   - Come identifico l'assenza del nodo?? (Rele non funzionante/non alimentato)
   - Acquisizione carico dopo accensione?? Dati carico in NVM!
   
   v1.0[07/05/15] - Create
*)
VAR CONSTANT
	MANUAL			: BYTE := 0;
	AUTOMATIC		: BYTE := 1;
	SCHEDULED		: BYTE := 2;
END_VAR
VAR_INPUT
	(* Settings *)
	ID				: BYTE;
	(* Controls *)
	CTRL_MODE		: BYTE;  (* 0 : MANUAL, (human) user manage the lux						->	HIGHEST PRIORITY
							    1 : AUTO, external device/sensor manage the lux				->	MID PRIORITY
							    2 : SCHEDULED, scheduled profile with crono manage the lux	->	LOWEST PRIORITY
							  *)

	(* Forced inputs *)
	LUX_ON_REQ		: BOOL; (* On request (Only "LUX_OFF_REQ" has highest priority) *)
	LUX_OFF_REQ		: BOOL; (* Off request (Highest priority over all other inputs/commands) *)

	(* External physical/software inputs *)
	CTRL_KEY		: BOOL := FALSE; (* External KEY control input *)
	KEY_PUSH		: BOOL := FALSE; (* 0: key as latch switch, 1: key as push-button, changes output state every time  *)
	CTRL_EXT_DS		: BOOL := FALSE; (* External DEVICE/SENSOR input *)
	CTRL_CRON		: BOOL := FALSE; (* External forced activation *)

	(* Conditional event *)
	CTRL_COND		: typ_Condition;
	CTRL_AUTO		: BOOL := TRUE;		(* 1: Lux managed by plc, 0: plc by-passed, managed by user	*)
	SINGLE_FEEDBACK	: BOOL;			 	(* Lux has its own feedback to control output status (state of art) or a general
										   feedback shared with other lux (loss of precision) *)

	(* Physical inputs (feedback) *)
	OUT_ST			: BOOL; (* Status feedback *)

END_VAR
VAR_IN_OUT
	WORKINGTIME		: DWORD; (* [sec] Internal working time counter *)
	POWERONCYCLES	: DWORD; (* Internal counter of power-on cycles *)
END_VAR
VAR_OUTPUT
	(* Physical outputs *)
	OUT_EN			: BOOL;	(* Control output *)
	(* Status *)
	Status_Log		: BYTE;
	Status_Vis 		: DWORD;
END_VAR
VAR
	InitOK			: BOOL;
	CTRL_MODE_Default: BYTE;
	Force			: BOOL := FALSE;		(* Force output to a value without considering its normal operation	*)

	KeyPress		: FLT_TIME 	:= (INITEV:=FALSE, TTAP:=T#5ms);
	AutoEn			: FLT_TAP := (INITEV:=FALSE);
	sOUT_EN			: FLT_EVENT;

	TickTimer		: TON := ( PT:=T#1s );
	chkOUT_ST		: FLT_TIME := ( TTAP:=T#5s);

	actualTime		: STRING;


END_VAR
Init();

(* Check if one or more conditional events are setted for this LUX *)
Condition();

IF LUX_OFF_REQ THEN OUT_EN := FALSE;
ELSIF LUX_ON_REQ OR NOT CTRL_AUTO THEN OUT_EN := TRUE;
ELSE
	(* Do actions according to acutal working mode *)
	CASE CTRL_MODE OF

		MANUAL:	(* Lux switching is managed by user	*)
	
			KeyPress(IN:=CTRL_KEY);
	
			IF KEY_PUSH THEN
				IF KeyPress.EVH THEN OUT_EN := NOT OUT_EN; END_IF	(* Key as push-button  ->  Toggle output *)
			ELSE
				IF KeyPress.EVH OR KeyPress.EVL THEN OUT_EN := CTRL_KEY; END_IF	(* Key as switch  ->  Open-Switch off
																									  Close-Switch on	*)
			END_IF

	
		AUTOMATIC:	(* Lux managed by an external device/sensor	*)

			KeyPress(IN:=CTRL_KEY);



			(* If a change in the key state has occured, switch to manual mode	*)
			IF KEY_PUSH THEN
				IF KeyPress.EVH THEN
					OUT_EN := NOT OUT_EN; 	(* Toggle output *)
					CTRL_MODE := MANUAL;
				END_IF
			ELSE
				IF KeyPress.EVH OR KeyPress.EVL THEN
					OUT_EN := CTRL_KEY;
					CTRL_MODE := MANUAL;
				END_IF
			END_IF

			(* These instructions are used to manage conditional event *)
			IF CTRL_MODE<>MANUAL THEN
				(* If not Forced keep automatic control *)
				IF NOT Force THEN
					(* Automatic mode *)
					AutoEn(IN:=CTRL_EXT_DS);
	
					(* IF AutoEn.EVH OR AutoEn.EVL THEN OUT_EN := NOT OUT_EN; END_IF *)
					IF AutoEn.EVH THEN OUT_EN := TRUE; END_IF
					IF AutoEn.EVL THEN OUT_EN := FALSE; END_IF
				END_IF
			END_IF

		SCHEDULED:
			(* Check if key has changed its state	*)
			KeyPress(IN:=CTRL_KEY);
	
			IF KEY_PUSH THEN
				IF KeyPress.EVH THEN
					OUT_EN := NOT OUT_EN; 	(* Toggle output *)
					CTRL_MODE := MANUAL;
				END_IF
			ELSE
				IF KeyPress.EVH OR KeyPress.EVL THEN
					OUT_EN := CTRL_KEY;
					CTRL_MODE := MANUAL;
				END_IF
			END_IF
	
			IF CTRL_MODE<>MANUAL THEN
				(* If not forced keep normal control *)
				IF NOT Force THEN
					(* Check if external control device has changed its state	*)
					AutoEn(IN:=CTRL_EXT_DS);
	
					IF AutoEn.EVH OR AutoEn.EVL THEN
						CTRL_MODE := AUTOMATIC;
						OUT_EN := NOT OUT_EN;
					END_IF
	
					IF CTRL_MODE<>AUTOMATIC THEN OUT_EN := CTRL_CRON;	END_IF	(* Scheduled mode	*)
				END_IF
			END_IF

	END_CASE
END_IF

(* Power on cycles and working time counters *)
Counters();

(* Check status feedback *)
IF SINGLE_FEEDBACK THEN chkOUT_ST(IN:=(OUT_ST<>OUT_EN));	(* External status feedback input available *)
ELSE chkOUT_ST(IN:=OUT_ST);						(* No external status feedback *)
END_IF
IF chkOUT_ST.EVH THEN LogEv(EL_Alarm,EO_LUX,ID,9,''); END_IF
IF chkOUT_ST.EVL THEN LogEv(EL_Log,EO_LUX,ID,1,''); END_IF

(* Status color *)
IF chkOUT_ST.OUT	THEN Status_Log:=2; (*Status_Vis:=COLOR_RED;*)
ELSE Status_Log:=0; Status_Vis:=SEL(OUT_EN,COLOR_GREEN_OFF,COLOR_GREEN);
END_IF
END_FUNCTION_BLOCK
ACTION AddLogData:
Logger.s1:=INSERT('&LUX=',BYTE_TO_STRING(ID),4);
IF ID<10 THEN Logger.s1:=INSERT(Logger.s1,'0',4); END_IF

Logger.s1:=CONCAT(Logger.s1,BOOL_TO_STRING(OUT_EN));			Logger.s1:=CONCAT(Logger.s1,';');
Logger.s1:=CONCAT(Logger.s1,DWORD_TO_STRING(WORKINGTIME));		Logger.s1:=CONCAT(Logger.s1,';');
Logger.s1:=CONCAT(Logger.s1,DWORD_TO_STRING(POWERONCYCLES));	Logger.s1:=CONCAT(Logger.s1,';');
Logger.s1:=CONCAT(Logger.s1,BYTE_TO_STRING(CTRL_MODE));			Logger.s1:=CONCAT(Logger.s1,';');
Logger.s1:=CONCAT(Logger.s1,BYTE_TO_STRING(Status_Log));
Logger.s1:=CONCAT(Logger.s1,';');
Logger.s1:=CONCAT(Logger.s1,SEL(LUX_ON_REQ,'0','100'));
Logger.s1:=CONCAT(Logger.s1,';');
Logger.s1:=CONCAT(Logger.s1,SEL(LUX_OFF_REQ,'0','100'));




ADDSTRING(ADR(Logger.TData), ADR(Logger.s1), Logger.TLen);
END_ACTION
ACTION Condition:
CASE CTRL_COND.Enable OF

	0:	(* NO CONDITION	*)
		;

	1:	(* BOOLEAN CONDITION - Trig On *)
		IF CTRL_COND.OnIN=CTRL_COND.OnValue THEN OUT_EN:=TRUE; END_IF

	2:	(* BOOLEAN CONDITION - Trig Off *)
		IF CTRL_COND.OffIN=CTRL_COND.OffValue THEN OUT_EN:=FALSE; END_IF

	3:	(* BOOLEAN CONDITION - Trig On and Off *)
		IF (OUT_EN=FALSE AND CTRL_COND.OnIN=CTRL_COND.OnValue) THEN OUT_EN:=TRUE; END_IF
		IF (OUT_EN=TRUE AND CTRL_COND.OffIN=CTRL_COND.OffValue) THEN OUT_EN:=FALSE; END_IF

	4: 	(* TIME of DAY - Trig On *)
		actualTime := MID(STR:=Sys.Time_LogString, LEN:=5, POS:=12);		(* Check if time of the day reached *)

		IF (OUT_EN=FALSE AND actualTime>=TOD_TO_STRING(CTRL_COND.OnTime)) THEN OUT_EN:=TRUE; END_IF

	5: 	(* TIME of DAY - Trig Off *)
		actualTime := MID(STR:=Sys.Time_LogString, LEN:=5, POS:=12);

		IF (OUT_EN=TRUE AND actualTime>=TOD_TO_STRING(CTRL_COND.OffTime)) THEN
			OUT_EN:= FALSE;
			Force := TRUE;
		END_IF

		IF actualTime>='08:00' THEN Force := FALSE; END_IF	(* Release force and restore normal working *)

END_CASE
END_ACTION
ACTION Counters:
(* Temporary energy counter *)
TickTimer(IN:=NOT TickTimer.Q);
IF (TickTimer.Q AND OUT_EN) THEN WORKINGTIME:=WORKINGTIME+1; END_IF

(* Generate status events *)
sOUT_EN(IN:=OUT_EN);
IF sOUT_EN.EVL THEN LogEv(EL_Log,EO_LUX,ID,2,''); END_IF
IF sOUT_EN.EVH THEN LogEv(EL_Log,EO_LUX,ID,3,''); POWERONCYCLES:=POWERONCYCLES+1; END_IF
END_ACTION
ACTION Init:
IF NOT InitOK THEN
	(* First time read the CTRL_MODE setted by the programmer in the global variables definition *)
	CTRL_MODE_Default := CTRL_MODE;
	InitOK := TRUE;
END_IF
END_ACTION
ACTION RestoreMode:
CTRL_MODE := CTRL_MODE_Default;

LUX_ON_REQ := FALSE;
LUX_OFF_REQ:= FALSE;
END_ACTION
ACTION StatReset:
(* Reset statistic counters *)
WORKINGTIME:=0;
POWERONCYCLES:=0;
END_ACTION

(* POU Plant_Objects/obj_MODBUS_FRER_QUBOH, ST *)
FUNCTION_BLOCK obj_MODBUS_FRER_QUBOH
(* === MODBUS ELECTRICITY CONTABILIZER ABB ===
   v1.0[20/08/15] - Versioning
*)
VAR CONSTANT
	WAIT_STATE		:	BYTE := 0;
	START_READ		:	BYTE := 1;
	READ_1			:	BYTE := 2;
	READ_2			:	BYTE := 3;
	READ_3			:	BYTE := 4;
	READ_4			:	BYTE := 5;
	READ_5			:	BYTE := 6;
	END_READ		:	BYTE := 7;
	WRITE_Q			:	BYTE := 8;
	READ_6			:	BYTE := 9;
	WRITE_ENABLE	:	BYTE := 10;

	ERROR_STATE		:	BYTE := 100;
END_VAR
VAR_INPUT
	ID				:	BYTE;
	Address			:	BYTE;

	Refresh_Period	: 	TIME:=t#1m;
	(* Controls *)
	Refresh_Auto	: 	BOOL:=TRUE; (* Enable automatic refresh *)
	Refresh_Now		:	BOOL; 	  (* Force an immediate refresh *)
END_VAR
VAR_IN_OUT
	ModBus		:	obj_MODBUS;
END_VAR
VAR_OUTPUT
	Status_Log	:	WORD;
	Status_Vis	:	DWORD;
END_VAR
VAR
	Data		:	typ_MODBUS_FRER_QUBOH;

	WH_3P		:	DWORD;		(* E-1 kWh *)
	VARH_3P		:	DWORD;		(* E-1 kVArh *)

	Q_Max		:	DWORD;

	dly 		: 	TON := (PT:=t#5s);
	state		: 	BYTE; 	(* Status *)
	retry		: 	BYTE;
END_VAR
CASE state OF

	WAIT_STATE: (* === Wait update signals *)
		dly(IN:=NOT (dly.Q OR Refresh_Now OR (NOT Refresh_Auto)));
		IF dly.Q OR Refresh_Now THEN
			dly.PT := Refresh_Period;
			Refresh_Now := FALSE;
			state := START_READ;
		END_IF

	START_READ:(* === Start update when MB is free *)
		IF NOT (ModBus.MB_Lock OR ModBus.MB_Start) THEN

			ModBus.MB_Lock := TRUE;
			ModBus.MB_Query.SlaveAddress := Address;
			ModBus.MB_Query.FunctionCode := 16#03;
			(* Start query *)
			ModBus.MB_Query.Read_StartAddress := 16#0100;
			ModBus.MB_Query.Read_Quantity := 32;
			ModBus.MB_Start := TRUE;

			state := READ_1;
		END_IF

	READ_1:
		IF NOT ModBus.MB_Start THEN
			IF ModBus.MB_MASTER.MB_Error<>MB_NO_ERROR OR ModBus.MB_Resp.Error<>0 THEN
				state := ERROR_STATE;
			ELSE
				(* Read response data *)
				COPY_32SWAP16(ADR(ModBus.MB_Resp.Data[0]), ADR(Data.V_L1N));
				COPY_32SWAP16(ADR(ModBus.MB_Resp.Data[2]), ADR(Data.V_L2N));
				COPY_32SWAP16(ADR(ModBus.MB_Resp.Data[4]), ADR(Data.V_L3N));
				COPY_32SWAP16(ADR(ModBus.MB_Resp.Data[6]), ADR(Data.V_L1L2));
				COPY_32SWAP16(ADR(ModBus.MB_Resp.Data[8]), ADR(Data.V_L2L3));
				COPY_32SWAP16(ADR(ModBus.MB_Resp.Data[10]), ADR(Data.V_L3L1));
				COPY_32SWAP16(ADR(ModBus.MB_Resp.Data[12]), ADR(Data.I_L1));
				COPY_32SWAP16(ADR(ModBus.MB_Resp.Data[14]), ADR(Data.I_L2));
				COPY_32SWAP16(ADR(ModBus.MB_Resp.Data[16]), ADR(Data.I_L3));
				COPY_32SWAP16(ADR(ModBus.MB_Resp.Data[18]), ADR(Data.FREQ));
				COPY_32SWAP16(ADR(ModBus.MB_Resp.Data[20]), ADR(Data.P_3P));
				COPY_32SWAP16(ADR(ModBus.MB_Resp.Data[22]), ADR(Data.Q_3P));
				COPY_32SWAP16(ADR(ModBus.MB_Resp.Data[24]), ADR(Data.PF_3P));
				COPY_32SWAP16(ADR(ModBus.MB_Resp.Data[26]), ADR(Data.WH_3P));
				COPY_32SWAP16(ADR(ModBus.MB_Resp.Data[28]), ADR(Data.VARH_3P));
				COPY_32SWAP16(ADR(ModBus.MB_Resp.Data[30]), ADR(Data.Multiplier));

				(* Evaluate energy according to read multiplier factor *)
				WH_3P := (Data.WH_3P * Data.Multiplier)/100;		(* Divided by 100 because read value is in Wh, we need E-1 kWh *)
				VARH_3P := (Data.VARH_3P * Data.Multiplier)/100;

				ModBus.MB_Query.Read_StartAddress := 16#0122;
				ModBus.MB_Query.Read_Quantity := 4;
				ModBus.MB_Start := TRUE;

				state := READ_2;
			END_IF
		END_IF

	READ_2:
		IF NOT ModBus.MB_Start THEN
			IF ModBus.MB_MASTER.MB_Error<>MB_NO_ERROR OR ModBus.MB_Resp.Error<>0 THEN
				state := ERROR_STATE;
			ELSE
				(* Read response data *)
				COPY_32SWAP16(ADR(ModBus.MB_Resp.Data[0]), ADR(Data.V_3P));
				COPY_32SWAP16(ADR(ModBus.MB_Resp.Data[2]), ADR(Data.I_3P));

				ModBus.MB_Query.Read_StartAddress := 16#012E;
				ModBus.MB_Query.Read_Quantity := 2;
				ModBus.MB_Start := TRUE;

				state := READ_3;
			END_IF
		END_IF

	READ_3:
		IF NOT ModBus.MB_Start THEN
			IF ModBus.MB_MASTER.MB_Error<>MB_NO_ERROR OR ModBus.MB_Resp.Error<>0 THEN
				state := ERROR_STATE;
			ELSE
				(* Read response data *)
				COPY_32SWAP16(ADR(ModBus.MB_Resp.Data[0]), ADR(Data.COS_3P));

				ModBus.MB_Query.Read_StartAddress := 16#0142;
				ModBus.MB_Query.Read_Quantity := 20;
				ModBus.MB_Start := TRUE;

				state := READ_4;
			END_IF
		END_IF

	READ_4:
		IF NOT ModBus.MB_Start THEN
			IF ModBus.MB_MASTER.MB_Error<>MB_NO_ERROR OR ModBus.MB_Resp.Error<>0 THEN
				state := ERROR_STATE;
			ELSE
				COPY_32SWAP16(ADR(ModBus.MB_Resp.Data[0]), ADR(Data.VA_3P));
				COPY_32SWAP16(ADR(ModBus.MB_Resp.Data[2]), ADR(Data.P_L1));
				COPY_32SWAP16(ADR(ModBus.MB_Resp.Data[4]), ADR(Data.P_L2));
				COPY_32SWAP16(ADR(ModBus.MB_Resp.Data[6]), ADR(Data.P_L3));
				COPY_32SWAP16(ADR(ModBus.MB_Resp.Data[8]), ADR(Data.Q_L1));
				COPY_32SWAP16(ADR(ModBus.MB_Resp.Data[10]), ADR(Data.Q_L2));
				COPY_32SWAP16(ADR(ModBus.MB_Resp.Data[12]), ADR(Data.Q_L3));
				COPY_32SWAP16(ADR(ModBus.MB_Resp.Data[14]), ADR(Data.VA_L1));
				COPY_32SWAP16(ADR(ModBus.MB_Resp.Data[16]), ADR(Data.VA_L2));
				COPY_32SWAP16(ADR(ModBus.MB_Resp.Data[18]), ADR(Data.VA_L3));

				ModBus.MB_Query.Read_StartAddress := 16#0156;
				ModBus.MB_Query.Read_Quantity := 22;
				ModBus.MB_Start := TRUE;

				state := READ_5;
			END_IF
		END_IF

	READ_5:
		IF NOT ModBus.MB_Start THEN
			IF ModBus.MB_MASTER.MB_Error<>MB_NO_ERROR OR ModBus.MB_Resp.Error<>0 THEN
				state := ERROR_STATE;
			ELSE
				COPY_32SWAP16(ADR(ModBus.MB_Resp.Data[0]), ADR(Data.PF_L1));
				COPY_32SWAP16(ADR(ModBus.MB_Resp.Data[2]), ADR(Data.PF_L2));
				COPY_32SWAP16(ADR(ModBus.MB_Resp.Data[4]), ADR(Data.PF_L3));
				COPY_32SWAP16(ADR(ModBus.MB_Resp.Data[6]), ADR(Data.COS_L1));
				COPY_32SWAP16(ADR(ModBus.MB_Resp.Data[8]), ADR(Data.COS_L2));
				COPY_32SWAP16(ADR(ModBus.MB_Resp.Data[10]), ADR(Data.COS_L3));
				COPY_32SWAP16(ADR(ModBus.MB_Resp.Data[12]), ADR(Data.P_3P_Max));
				COPY_32SWAP16(ADR(ModBus.MB_Resp.Data[14]), ADR(Data.P_3P_Avg));
				COPY_32SWAP16(ADR(ModBus.MB_Resp.Data[16]), ADR(Data.I_L1_Max));
				COPY_32SWAP16(ADR(ModBus.MB_Resp.Data[18]), ADR(Data.I_L2_Max));
				COPY_32SWAP16(ADR(ModBus.MB_Resp.Data[20]), ADR(Data.I_L3_Max));

				ModBus.MB_Query.Read_StartAddress := 16#01A6;
				ModBus.MB_Query.Read_Quantity := 2;
				ModBus.MB_Start := TRUE;

				state := END_READ;
			END_IF
		END_IF

	END_READ:
		IF NOT ModBus.MB_Start THEN
			IF ModBus.MB_MASTER.MB_Error<>MB_NO_ERROR OR ModBus.MB_Resp.Error<>0 THEN
				state := ERROR_STATE;
			ELSE
				COPY_32SWAP16(ADR(ModBus.MB_Resp.Data[0]), ADR(Data.Q_3P_Max));

				ModBus.MB_Query.Write_StartAddress := 16#200;
				ModBus.MB_Query.FunctionCode := 16#10;
				ModBus.MB_Query.Write_Quantity := 2;
				ModBus.MB_Query.Write_Data[0] := 16#0000;
				ModBus.MB_Query.Write_Data[1] := 16#00A5;
				ModBus.MB_Start := TRUE;

				state := WRITE_ENABLE;
			END_IF
		END_IF

	WRITE_ENABLE:
		IF NOT ModBus.MB_Start THEN
			IF ModBus.MB_MASTER.MB_Error<>MB_NO_ERROR OR ModBus.MB_Resp.Error<>0 THEN
				state := ERROR_STATE;
			ELSE
				COPY_32SWAP16(ADR(ModBus.MB_Resp.Data[0]), ADR(Data.Q_3P_Max));

				ModBus.MB_Query.Write_StartAddress := 16#01A6;
				ModBus.MB_Query.FunctionCode := 16#10;
				ModBus.MB_Query.Write_Quantity := 2;
				ModBus.MB_Query.Write_Data[0] := 16#0000;
				ModBus.MB_Query.Write_Data[1] := 16#0000;
				ModBus.MB_Start := TRUE;

				state := WRITE_Q;
			END_IF
		END_IF

	WRITE_Q:
		IF NOT ModBus.MB_Start THEN
			IF ModBus.MB_MASTER.MB_Error<>MB_NO_ERROR OR ModBus.MB_Resp.Error<>0 THEN
				state := ERROR_STATE;
			ELSE
				ModBus.MB_Query.Read_StartAddress := 16#01A6;
				ModBus.MB_Query.FunctionCode := 16#03;
				ModBus.MB_Query.Read_Quantity := 2;

				ModBus.MB_Start := TRUE;
				state := READ_6;
			END_IF
		END_IF

	READ_6:
		IF NOT ModBus.MB_Start THEN
			IF ModBus.MB_MASTER.MB_Error<>MB_NO_ERROR OR ModBus.MB_Resp.Error<>0 THEN
				state := ERROR_STATE;
			ELSE
				COPY_32SWAP16(ADR(ModBus.MB_Resp.Data[0]), ADR(Q_Max));
				(* Signal event *)
				(*IF Status_Log<>0 THEN
					LogEv(EL_Log,EO_ANZ,ID,1,'');
				END_IF*)

				(* Update status *)
				Status_Log:=0;

				ModBus.MB_Lock := FALSE;
				retry := 0;
				state := WAIT_STATE;
			END_IF
		END_IF

	ERROR_STATE: (* === Check MODBUS error *)
			(* Release MODBUS *)
			MODBUS.MB_Lock:=FALSE;

			(* Retries *)
			retry:=retry+1;

			IF retry>3 THEN
				retry:=0;
				(* Signal event *)
				IF Status_Log<>2 THEN
					LogEv(EL_Alarm,EO_ANZ,ID,2,SEL(ModBus.MB_MASTER.MB_Error<>0,'0','1'));
				END_IF
				(* Update status *)
				Status_Log:=2;
			END_IF

			state := WAIT_STATE;

END_CASE

IF Status_Log=2 THEN Status_Vis := COLOR_RED;
ELSE Status_Vis := COLOR_GREEN;
END_IF
END_FUNCTION_BLOCK
ACTION AddLogData:
Logger.s1:=INSERT('&ANZ=',BYTE_TO_STRING(ID),4);
IF ID<10 THEN Logger.s1:=INSERT(Logger.s1,'0',4); END_IF

Logger.s1:=CONCAT(Logger.s1,DWORD_TO_STRING(Data.V_L1N/1000));		Logger.s1:=CONCAT(Logger.s1,';');
Logger.s1:=CONCAT(Logger.s1,DWORD_TO_STRING(Data.V_L2N/1000));		Logger.s1:=CONCAT(Logger.s1,';');
Logger.s1:=CONCAT(Logger.s1,DWORD_TO_STRING(Data.V_L3N/1000));		Logger.s1:=CONCAT(Logger.s1,';');
Logger.s1:=CONCAT(Logger.s1,DWORD_TO_STRING(Data.V_L1L2/1000));		Logger.s1:=CONCAT(Logger.s1,';');
Logger.s1:=CONCAT(Logger.s1,DWORD_TO_STRING(Data.V_L2L3/1000));		Logger.s1:=CONCAT(Logger.s1,';');
Logger.s1:=CONCAT(Logger.s1,DWORD_TO_STRING(Data.V_L3L1/1000));		Logger.s1:=CONCAT(Logger.s1,';');

Logger.s1:=CONCAT(Logger.s1,DWORD_TO_STRING(Data.FREQ));		Logger.s1:=CONCAT(Logger.s1,';');

Logger.s1:=CONCAT(Logger.s1,DWORD_TO_STRING(Data.I_L1));		Logger.s1:=CONCAT(Logger.s1,';');
Logger.s1:=CONCAT(Logger.s1,DWORD_TO_STRING(Data.I_L2));		Logger.s1:=CONCAT(Logger.s1,';');
Logger.s1:=CONCAT(Logger.s1,DWORD_TO_STRING(Data.I_L3));		Logger.s1:=CONCAT(Logger.s1,';');
Logger.s1:=CONCAT(Logger.s1,DWORD_TO_STRING(Data.I_L1_Max)); 	Logger.s1:=CONCAT(Logger.s1,';');
Logger.s1:=CONCAT(Logger.s1,DWORD_TO_STRING(Data.I_L2_Max)); 	Logger.s1:=CONCAT(Logger.s1,';');
Logger.s1:=CONCAT(Logger.s1,DWORD_TO_STRING(Data.I_L3_Max)); 	Logger.s1:=CONCAT(Logger.s1,';');

Logger.s1:=CONCAT(Logger.s1,DINT_TO_STRING(Data.PF_L1));		Logger.s1:=CONCAT(Logger.s1,';');
Logger.s1:=CONCAT(Logger.s1,DINT_TO_STRING(Data.PF_L2));		Logger.s1:=CONCAT(Logger.s1,';');
Logger.s1:=CONCAT(Logger.s1,DINT_TO_STRING(Data.PF_L3));		Logger.s1:=CONCAT(Logger.s1,';');

Logger.s1:=CONCAT(Logger.s1,DWORD_TO_STRING(Data.P_3P));		Logger.s1:=CONCAT(Logger.s1,';');
Logger.s1:=CONCAT(Logger.s1,DWORD_TO_STRING(Data.P_3P_Avg)); 	Logger.s1:=CONCAT(Logger.s1,';');
Logger.s1:=CONCAT(Logger.s1,DWORD_TO_STRING(Data.P_3P_Max)); 	Logger.s1:=CONCAT(Logger.s1,';');

Logger.s1:=CONCAT(Logger.s1,DINT_TO_STRING(Data.Q_3P));			Logger.s1:=CONCAT(Logger.s1,';');
Logger.s1:=CONCAT(Logger.s1,DINT_TO_STRING(Data.Q_3P_Max));		Logger.s1:=CONCAT(Logger.s1,';');

Logger.s1:=CONCAT(Logger.s1,DWORD_TO_STRING(WH_3P));			Logger.s1:=CONCAT(Logger.s1,';');
Logger.s1:=CONCAT(Logger.s1,DWORD_TO_STRING(VARH_3P));			Logger.s1:=CONCAT(Logger.s1,';');

Logger.s1:=CONCAT(Logger.s1,WORD_TO_STRING(Status_Log));
ADDSTRING(ADR(Logger.TData), ADR(Logger.s1), Logger.TLen);
END_ACTION

(* POU Plant_Objects/obj_MODBUS_TCP, ST *)
FUNCTION_BLOCK obj_MODBUS_TCP
(* === MODBUS-TCP PROTOCOL INTERFACE ===
   v1.0[10/06/15] - Create
*)
VAR CONSTANT
	VARS_Max	: BYTE := 32;
END_VAR
VAR_INPUT
	(* Settings *)
	ID			: BYTE;
	IP			: STRING;
	PORT		: WORD:=502;
	(* Interface *)
	MB_MASTER	: ETHERNET_MODBUSMASTER_TCP;
	MB_READBUF	: ARRAY [0..128] OF WORD;
	MB_WRITEBUF : ARRAY [0..128] OF WORD;
	MB_Start	: BOOL;
	MB_Lock		: BOOL;
	(* Variables management *)
	VARS_En		: BOOL;
	VARS		: ARRAY [0..VARS_Max] OF typ_MODBUS_VAR;
	VARS_Check	: BOOL;
	VARS_Alarm	: BOOL;
	(* Variables allocation *)
	VAR_Pointer : POINTER TO ARRAY[0..99] OF WORD;
	VAR_Cfg		: POINTER TO typ_MODBUS_VAR;
END_VAR
VAR_OUTPUT
	(* Status *)
	Status_Log	: BYTE;
	Status_Vis	: DWORD;
END_VAR
VAR
	sta         : BYTE :=0;
	i			: BYTE;
	j			: BYTE;
	Alarm		: FLT_EVENT := (INITEV:=FALSE);

	VarTmr		: TON := (PT:=T#1s);
	VarSta		: BYTE; (* Status *)
	VarCnt		: BYTE; (* Scan counter *)
	VarRetry	: BYTE;
	VarAlarm	: BYTE; (* Last variable with errors *)
END_VAR
MB_MASTER( strIP_ADDRESS:=IP, wPORT:=PORT, tTIME_OUT:=T#750MS, (*xCONNECT:=TRUE,*)
		   ptREAD_DATA:=ADR(MB_READBUF), ptSEND_DATA:=ADR(MB_WRITEBUF), xSEND:=MB_Start );

IF sta=0 THEN
	MB_MASTER.xCONNECT:=TRUE;
	sta:=1;
END_IF

(* Process variable management *)
IF VARS_En THEN VARS_Process(); END_IF

(* Check status *)
Alarm(IN:=(MB_MASTER.wERROR<>0));
IF Alarm.EVH THEN
	LogEv(SEL(MB_MASTER.wERROR>0,EL_Wrn,EL_Alarm),EO_MODBUS_TCP,ID,1,WORD_TO_STRING(MB_MASTER.wERROR));
END_IF
IF Alarm.EVL THEN
	LogEv(EL_Log,EO_MODBUS_TCP,ID,2,'');
END_IF

(* Log/visu status *)
   IF Alarm.IN   THEN Status_Log:=2; Status_Vis:=COLOR_RED;
ELSIF Vars_Alarm THEN Status_Log:=1; Status_Vis:=COLOR_YELLOW;
  				 ELSE Status_Log:=0; Status_Vis:=COLOR_GREEN;
END_IF
END_FUNCTION_BLOCK
ACTION VAR_Search:
(* Search VAR with specific pointer if not found return first free VAR
	[Last VAR is not active... used as safe area...] 
*)
j:=VARS_Max;
FOR i := 0 TO VARS_Max-1 DO
	IF VARS[i].Variable=0 AND j>i THEN j:=i; END_IF
	IF VARS[i].Variable=VAR_Pointer THEN
		VAR_Cfg:=ADR(VARS[i]);
		RETURN;
	END_IF
END_FOR
VAR_Cfg:=ADR(VARS[j]);
END_ACTION
ACTION VARS_Process:
(* Update var timers *)
VarTmr(IN:=(NOT VarTmr.Q));
IF VarTmr.Q THEN
	FOR i := 0 TO VARS_Max DO
		IF VARS[i].Refresh_Cnt>0 THEN VARS[i].Refresh_Cnt:=VARS[i].Refresh_Cnt-1; END_IF
	END_FOR
	VARS_Check:=TRUE;
END_IF


(* Process status *)
CASE VarSta OF
	0: (* === Init *)
		VarCnt:=0;
		VarSta:=1;

	1: (* === Wait check signal *)
		IF VARS_Check THEN
			VARS_Check:=FALSE;
			VarCnt:=0;
			VarSta:=2;
		END_IF

	2: (* === Check loop *)
		IF NOT (MB_Lock OR MB_Start) THEN
			WHILE VarCnt<=(VARS_Max-1) AND VarSta=2 DO
				(* Check only active vars *)
				IF VARS[VarCnt].Variable<>0 THEN
					(* Check var auto-refresh on timer checks *)
					IF VARS[VarCnt].Refresh_Time>0 AND VARS[VarCnt].Refresh_Cnt=0 THEN
						VARS[VarCnt].Refresh_Cnt:=VARS[VarCnt].Refresh_Time;
						VarSta:=3;
					END_IF
					(* Check refresh for change or request *)
					CASE VARS[VarCnt].FunCode OF
						5,6,15,16: (* Write functions *)
							IF VARS[VarCnt].Variable_Size=1 THEN
								IF VARS[VarCnt].Variable^<>VARS[VarCnt].Variable_Mirror THEN
									VARS[VarCnt].Variable_Mirror:=VARS[VarCnt].Variable^;
									VarSta:=3;
								END_IF
							ELSE
								IF VARS[VarCnt].Variable_Mirror<>0 THEN
									VARS[VarCnt].Variable_Mirror:=0;
									VarSta:=3;
								END_IF
							END_IF
						1,2,3,4: (* Write functions *)
							IF VARS[VarCnt].Variable_Mirror<>0 THEN
								VARS[VarCnt].Variable_Mirror:=0;
								VarSta:=3;
							END_IF
					END_CASE
				END_IF
				(* Process query *)
				IF VarSta=3 THEN
					MB_Lock:=TRUE;
					MB_MASTER.bUNIT_ID:=VARS[VarCnt].SlaveAddress;
					MB_MASTER.bFUNCTION_CODE:=VARS[VarCnt].FunCode;
					CASE VARS[VarCnt].FunCode OF
						16#5,16#6,16#F,16#10:
							MB_MASTER.wREAD_ADDRESS:=0;
							MB_MASTER.wREAD_QUANTITY:=0;
							MB_MASTER.wWRITE_ADDRESS:=VARS[VarCnt].FunAddress;
							MB_MASTER.wWRITE_QUANTITY:=VARS[VarCnt].Variable_Size;
							IF VARS[VarCnt].Variable_Size=200 THEN
								COPY_32SWAP16(VARS[VarCnt].Variable, ADR(MB_WRITEBUF));
							ELSIF VARS[VarCnt].Variable_Size>1 THEN
								MEMCPY(VARS[VarCnt].Variable, ADR(MB_WRITEBUF), 2*VARS[VarCnt].Variable_Size);
							ELSE
								MB_WRITEBUF[0]:=VARS[VarCnt].Variable^;
							END_IF
						16#1,16#2,16#3,16#4:
							MB_MASTER.wREAD_ADDRESS:=VARS[VarCnt].FunAddress;
							IF VARS[VarCnt].Variable_Size=200 THEN MB_MASTER.wREAD_QUANTITY:=2; ELSE
							  MB_MASTER.wREAD_QUANTITY:=VARS[VarCnt].Variable_Size;
							END_IF
							MB_MASTER.wWRITE_ADDRESS:=0;
							MB_MASTER.wWRITE_QUANTITY:=0;
					END_CASE
					VarRetry:=0;
					MB_Start:=TRUE;
				ELSE
					VarCnt:=VarCnt+1;
				END_IF
			END_WHILE
			(* Check loop completed -> no actions *)
			IF VarSta=2 THEN VarSta:=1; END_IF
		END_IF

	3: (* === Wait & process MB response *)
		IF NOT MB_Start THEN
			IF MB_MASTER.wERROR=0 THEN
				CASE VARS[VarCnt].FunCode OF
					1,2,3,4:
						IF VARS[VarCnt].Variable_Size=200 THEN
							COPY_32SWAP16(ADR(MB_READBUF), VARS[VarCnt].Variable);
						ELSIF VARS[VarCnt].Variable_Size>1 THEN
							MEMCPY(ADR(MB_READBUF), VARS[VarCnt].Variable, 2*VARS[VarCnt].Variable_Size);
						ELSE
							VARS[VarCnt].Variable^:=MB_READBUF[0];
						END_IF
				END_CASE
				MB_Lock:=FALSE;
				(* Signal error recovery *)
				IF VARS_Alarm=TRUE AND VarCnt=VarAlarm THEN
					LogEv(EL_Wrn,EO_MODBUS_TCP,ID,5,'');
					VARS_Alarm:=FALSE;
				END_IF
				(* Next var *)
				VarCnt:=VarCnt+1;
				VarSta:=2;
			ELSE
				IF VarRetry<10 THEN
					VarRetry:=VarRetry+1;
					MB_Start:=TRUE;
				ELSE
					MB_Lock:=FALSE;
					(* Signal error *)
					IF VARS_Alarm=FALSE THEN
						LogEv(EL_Wrn,EO_MODBUS_TCP,ID,3,WORD_TO_STRING(MB_MASTER.wERROR));
						VARS_Alarm:=TRUE;
						VarAlarm:=VarCnt-1;
					END_IF
					(* Next var *)
					VarCnt:=VarCnt+1;
					VarSta:=2;
				END_IF
			END_IF
		END_IF

ELSE
	VarSta:=0;
END_CASE
END_ACTION

(* POU Plant_Objects/obj_ZTHL, ST *)
FUNCTION_BLOCK obj_ZTHL
(* === ZIGBEE AMBIENT SENSORS MT-200 ===
   v1.0[07/05/05] - Create
*)
VAR CONSTANT
	(* States *)
	WAIT_STATE			:	BYTE := 0;
	STATUS_REQUEST		:	BYTE := 1;
	LQI_REQUEST			:	BYTE := 2;
	MEAS_REQUEST		:	BYTE := 3;
	END_READ			:	BYTE := 4;
	ERROR_STATE			:	BYTE := 100;

	LQI_Threshold		:	WORD := 100;		(* Zigbee link quality minimum value *)
	LowBattVoltage		:	WORD := 270;		(* Battery is considered low when reaches 1.35V each *)
END_VAR
VAR_INPUT
	(* Settings *)
	ID				: BYTE;
	Address			: BYTE;

	Refresh_Period	: TIME:=t#5m;
	(* Controls *)
	Refresh_Auto	: BOOL:=TRUE; (* Enable automatic refresh *)
	Refresh_Now		: BOOL; 	  (* Force an immediate refresh *)

	(* Limits *)
	Tmin			: INT := 0;
	Tmax			: INT := 400;
END_VAR
VAR_IN_OUT
	(* Interface *)
	MODBUS			: obj_MODBUS_TCP;
END_VAR
VAR_OUTPUT
	NodeStatus		: WORD;
	OUT_TEMP		: INT;	(* Temperatura misurata [°C/10] *)
	OUT_HYGRO		: INT;	(* Umidità misurata [%] *)
	OUT_LUX			: INT;	(* Luce misurata [lux] *)
	OUT_VBATT		: INT;	(* Tensione misurata dalla batteria [V/100] *)

	OUT_LQI			: BYTE;

	ERR				: BOOL;

	fTemp			: BOOL;

	(* Status *)
	Status_Log		: BYTE;
	Status_Vis 		: DWORD;
END_VAR
VAR
	dly 	 		: TON := (PT:=t#5s);

	sta				: BYTE;
	retry	 		: BYTE;

	OldNodeStatus	: WORD;
	fLQI			: BOOL;
	fBatt			: BOOL;
	Quality			: FLT_EVENT;
	Battery			: FLT_EVENT;
	Temperature		: FLT_EVENT := (INITEV:=FALSE);
	Alarm			: FLT_EVENT;

	StatusOK		: BYTE;			(* 0: Status OK, >=1: Alarm and/or warning		Incremented by 1 when Alarm or Wrn occurs,
																					decremented by 1 when restored	*)
END_VAR
CASE sta OF
	WAIT_STATE: (* === Wait update signals *)
		dly(IN:=NOT (dly.Q OR Refresh_Now OR (NOT Refresh_Auto)));
		IF dly.Q OR Refresh_Now THEN
			dly.PT:=Refresh_Period;
			Refresh_Now:=FALSE;
			(*sta:=STATUS_REQUEST;*)
			sta:=LQI_REQUEST;
		END_IF

	STATUS_REQUEST:	(* Node status *)
		IF NOT (MODBUS.MB_Lock OR MODBUS.MB_Start) THEN
			MODBUS.MB_Lock:=TRUE;
			MODBUS.ID:=ID;
			MODBUS.MB_MASTER.bUNIT_ID := Address;
			MODBUS.MB_MASTER.bFUNCTION_CODE:=16#03;
			MODBUS.MB_MASTER.wREAD_ADDRESS:=16#0D;
			MODBUS.MB_MASTER.wREAD_QUANTITY:=16#1;
			MODBUS.MB_Start:=TRUE;
			sta:=LQI_REQUEST;
		END_IF

	LQI_REQUEST:	(* Link quality *)
		IF NOT MODBUS.MB_Start THEN
			IF MODBUS.MB_MASTER.wERROR<>MB_NO_ERROR THEN
				sta:=ERROR_STATE;
			ELSE
				NodeStatus	:=	MODBUS.MB_READBUF[0];

				MODBUS.ID:=ID;
				MODBUS.MB_MASTER.bUNIT_ID := Address;
				MODBUS.MB_MASTER.bFUNCTION_CODE:=16#03;
				MODBUS.MB_MASTER.wREAD_ADDRESS:=16#01;
				MODBUS.MB_MASTER.wREAD_QUANTITY:=16#1;
				MODBUS.MB_Start:=TRUE;

				sta:=MEAS_REQUEST;
			END_IF
		END_IF

	MEAS_REQUEST:	(* Measurements *)
		IF NOT MODBUS.MB_Start THEN
			IF MODBUS.MB_MASTER.wERROR<>MB_NO_ERROR THEN
				sta:=ERROR_STATE;
			ELSE

				OUT_LQI	:=	WORD_TO_BYTE(MODBUS.MB_READBUF[0]);

				MODBUS.ID:=ID;
				MODBUS.MB_MASTER.bUNIT_ID := Address;
				MODBUS.MB_MASTER.bFUNCTION_CODE:=16#03;
				MODBUS.MB_MASTER.wREAD_ADDRESS:=16#14;
				MODBUS.MB_MASTER.wREAD_QUANTITY:=16#5;
				MODBUS.MB_Start:=TRUE;

				sta:=END_READ;
			END_IF
		END_IF

	END_READ:	IF NOT MODBUS.MB_Start THEN
			IF MODBUS.MB_MASTER.wERROR<>MB_NO_ERROR THEN
				sta:=ERROR_STATE;
			ELSE
				OUT_TEMP	:=	WORD_TO_INT(MODBUS.MB_READBUF[0]);
				OUT_HYGRO	:=	WORD_TO_INT(MODBUS.MB_READBUF[1]);
				OUT_LUX		:=	WORD_TO_INT(MODBUS.MB_READBUF[2]);
				OUT_VBATT	:=	WORD_TO_INT(MODBUS.MB_READBUF[3]);
				sta:=WAIT_STATE;
				MODBUS.MB_Lock:=FALSE;
			END_IF
		END_IF

	ERROR_STATE:
			MODBUS.MB_Lock:=FALSE;
			(* Retries *)
			retry:=retry+1;
			IF retry>3 THEN
				retry:=0;
				IF Status_Log<>2 THEN
					LogEv(EL_Alarm,EO_ZTHL,ID,4,'');
				END_IF
				Status_Log:=2;
				Status_Vis:=COLOR_RED;
			END_IF
			sta:=WAIT_STATE;

ELSE
			sta:=WAIT_STATE;
END_CASE

(* Check Status *)
(*
IF NodeStatus <> OldNodeStatus THEN
	IF NodeStatus = 3 THEN
		LogEv(EL_Alarm,EO_ZTHL,ID,3,'');
		Status_Log:=2;
	ELSE
		Status_Log:=0;
	END_IF

	OldNodeStatus := NodeStatus;
END_IF*)

(* Check Link quality *)

IF OUT_LQI < LQI_Threshold THEN
	fLQI := TRUE;
	ERR := TRUE;
ELSE
	fLQI := FALSE;
	ERR := FALSE;
END_IF

Quality(IN:=fLQI);

IF Quality.EVL THEN
	LogEv(SEL(OUT_LQI<>0,EL_Alarm,EL_Wrn),EO_ZTHL,ID,SEL(OUT_LQI<>0,7,2),WORD_TO_STRING(OUT_LQI));
	Status_Log := SEL(OUT_LQI<>0,2,1);
	StatusOK := StatusOK + 1;
END_IF

IF Quality.EVH THEN StatusOK := SEL(StatusOK=0, StatusOK-1, 0); END_IF

(* If probe (node) is present proceed checking other warnings, otherwise don't transmit anything *)
IF OUT_LQI <> 0 THEN

	(* Check battery voltage *)


	IF OUT_VBATT < LowBattVoltage THEN fBatt := TRUE;
	ELSE fBatt := FALSE;
	END_IF


	Battery(IN:=fBatt);

	IF Battery.EVH  THEN
		LogEv(EL_Wrn,EO_ZTHL,ID,6,' ');
		StatusOK := StatusOK + 1;
	END_IF

	IF Battery.EVL THEN StatusOK := SEL(StatusOK=0, StatusOK-1, 0); END_IF

	(* Check Node temperature *)
	IF OUT_TEMP < Tmin OR OUT_TEMP > Tmax THEN
		fTemp := TRUE;
		ERR := TRUE;
	ELSE
		fTemp := FALSE;
		ERR := FALSE;
	END_IF

	Temperature(IN:=fTemp);

	IF Temperature.EVH THEN
		LogEv(EL_Wrn,EO_ZTHL,ID,5,INT_TO_STRING(OUT_TEMP));
		Status_Log := 1;
		StatusOK := StatusOK + 1;
	END_IF

	IF Temperature.EVL THEN StatusOK := SEL(StatusOK=0, StatusOK-1, 0); END_IF

END_IF

Alarm(IN:=(StatusOK=0));

IF Alarm.EVH THEN
	Status_Log := 0;
	LogEv(EL_Log,EO_ZTHL,ID,1,'');
END_IF

IF Status_Log = 2 THEN Status_Vis := COLOR_RED;
ELSIF Status_Log = 1 THEN Status_Vis := COLOR_YELLOW;
ELSE Status_Vis := COLOR_GREEN;
END_IF
END_FUNCTION_BLOCK
ACTION AddLogData:
Logger.s1:=INSERT('&ZTHL=',BYTE_TO_STRING(ID),5);
IF ID<10 THEN Logger.s1:=INSERT(Logger.s1,'0',5); END_IF

Logger.s1:=CONCAT(Logger.s1,BYTE_TO_STRING(OUT_LQI));			Logger.s1:=CONCAT(Logger.s1,';');
Logger.s1:=CONCAT(Logger.s1,INT_TO_STRING(OUT_TEMP ));			Logger.s1:=CONCAT(Logger.s1,';');
Logger.s1:=CONCAT(Logger.s1,INT_TO_STRING(OUT_HYGRO ));			Logger.s1:=CONCAT(Logger.s1,';');
Logger.s1:=CONCAT(Logger.s1,INT_TO_STRING(OUT_LUX));			Logger.s1:=CONCAT(Logger.s1,';');
Logger.s1:=CONCAT(Logger.s1,INT_TO_STRING(OUT_VBATT));			Logger.s1:=CONCAT(Logger.s1,';');

Logger.s1:=CONCAT(Logger.s1,BYTE_TO_STRING(Status_Log));
ADDSTRING(ADR(Logger.TData), ADR(Logger.s1), Logger.TLen);
END_ACTION

(* POU PLC_WDT, ST *)
FUNCTION PLC_WDT: DWORD VAR_INPUT dwEvent: DWORD; dwFilter: DWORD; dwOwner: DWORD; END_VAR
LogEv(EL_AlarmStop,EO_SYS,1,10,'Watchdog');
END_FUNCTION

(* POU Utils Functions/RAWTOHEXSTR, ST *)
FUNCTION RAWTOHEXSTR : STRING(128)
VAR_INPUT
	pData: POINTER TO BYTE;
	DataLen: BYTE;
END_VAR
VAR
	pt: POINTER TO BYTE;
	xl: BYTE;
END_VAR
pt:=ADR(RAWTOHEXSTR);

xl:=2;

WHILE DataLen>0 AND xl<128 DO

	pt^ := (pData^ / 16#10) + 48 + (((pData^ / 16#10)/10)*7);
	pt:=pt+1;
	pt^ := (pData^ AND 16#0F)  + 48 + (((pData^ AND 16#0F)/10)*7);
	pt:=pt+1;

	xl:=xl+2;

	DataLen:=DataLen-1;
	pData:=pData+1;

END_WHILE

pt^:=0;
END_FUNCTION

(* POU Utils Functions/RESET_ARRAY, ST *)
FUNCTION RESET_ARRAY : BOOL
VAR_INPUT
	pData	:	POINTER TO WORD;
	Size	:	BYTE;
END_VAR
VAR
	i	:	BYTE := 0;
END_VAR
WHILE i<Size DO

	pData^ := 0;
	pData := pData + 1;
	i := i + 1;

END_WHILE
END_FUNCTION

(* POU Utils/RTC_Update, ST *)
FUNCTION RTC_Update : BOOL
VAR
	T: DT;
	TS: STRING;
	TS2: STRING;
	Hour: BYTE;
	Minute: BYTE;
END_VAR
(* Get RTC time *)
T:=SysRtcGetTime(TRUE);
Sys.Time_CT_DT:=T;
(* Calculate variables *)
TS:=DT_TO_STRING(T);
Sys.Time_LogString:=DELETE(STR:=TS, LEN:=3, POS:=1);
TS2:=MID(STR:=TS, LEN:=4, POS:= 4); Sys.Time_Year 	:=STRING_TO_WORD(TS2);
TS2:=MID(STR:=TS, LEN:=2, POS:= 9); Sys.Time_Month	:=STRING_TO_BYTE(TS2);
TS2:=MID(STR:=TS, LEN:=2, POS:=12); Sys.Time_Day  	:=STRING_TO_BYTE(TS2);
Sys.Time_CT_Day:=(32*(Sys.Time_Month-1)+Sys.Time_Day-1);
TS2:=MID(STR:=TS, LEN:=2, POS:=15); Hour			:=STRING_TO_BYTE(TS2);
TS2:=MID(STR:=TS, LEN:=2, POS:=18); Minute		 	:=STRING_TO_BYTE(TS2);
Sys.Time_CT_Quarter:=Hour*4+(Minute/15);
END_FUNCTION

(* POU Utils Functions/SHIFT_ARRAY, ST *)
FUNCTION SHIFT_ARRAY : BOOL
VAR_INPUT
	pData	:	POINTER TO ARRAY [1..2] OF WORD;
	Size	:	BYTE;
END_VAR
VAR
	pNew	:	POINTER TO WORD;
	i		:	BYTE;
END_VAR
(* Shift right *)
FOR i:=1 TO (Size-1) BY 1 DO

	(*pNew := pData + 1;*)
	pData^[i] := pData^[i+1];
	(*pData := pData + 1;*)

END_FOR
END_FUNCTION

(* POU Utils Functions/TONOF, ST *)
FUNCTION_BLOCK TONOF
VAR_INPUT
	IN		: BOOL;
	PT_ON	: TIME; (* time to pass, before OUT is set *)
	PT_OF	: TIME; (* time to pass, before OUT is reset *)
END_VAR
VAR_OUTPUT
	OUT		: BOOL;
END_VAR
VAR
	timer	: TON;
END_VAR
IF IN<>OUT THEN
	timer(IN:=TRUE,PT:=SEL(IN,PT_OF,PT_ON));
	IF timer.Q THEN OUT:=IN; END_IF
ELSE
	timer(IN:=FALSE);
END_IF
END_FUNCTION_BLOCK

(* Visualisation PLC_VISU
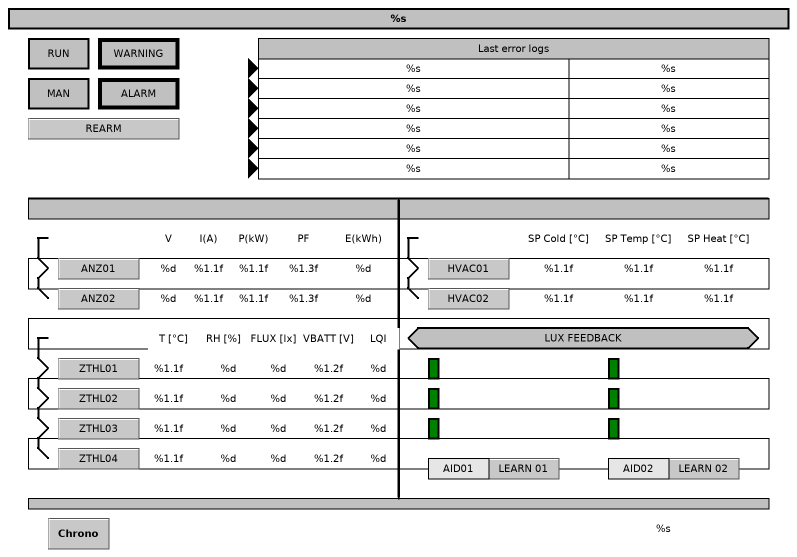
rectangle at (10,0)-(791,21): text "%s"; shows .Plant_NAME
rounded rectangle at (30,30)-(91,61): text "RUN"; alarm colour if NOT Mode_Manual; runs INTERN ASSIGN Mode_Manual:=(FALSE)
rounded rectangle at (30,70)-(91,101): text "MAN"; alarm colour if Mode_Manual; runs INTERN ASSIGN Mode_Manual:=(TRUE)
rectangle at (570,50)-(771,71): text "%s"; shows Sys.LastLogs_Msg[0]
polygon at (250,150)-(260,170): invisible if Sys.LastLogs_Idx<>0
rectangle at (570,70)-(771,91): text "%s"; shows Sys.LastLogs_Msg[1]
polygon at (250,50)-(260,70): invisible if Sys.LastLogs_Idx<>1
rectangle at (570,90)-(771,111): text "%s"; shows Sys.LastLogs_Msg[2]
polygon at (250,70)-(260,90): invisible if Sys.LastLogs_Idx<>2
rectangle at (570,110)-(771,131): text "%s"; shows Sys.LastLogs_Msg[3]
polygon at (250,90)-(260,110): invisible if Sys.LastLogs_Idx<>3
rectangle at (570,130)-(771,151): text "%s"; shows Sys.LastLogs_Msg[4]
polygon at (250,110)-(260,130): invisible if Sys.LastLogs_Idx<>4
rectangle at (570,150)-(771,171): text "%s"; shows Sys.LastLogs_Msg[5]
polygon at (250,130)-(260,150): invisible if Sys.LastLogs_Idx<>5
rectangle at (260,50)-(571,71): text "%s"; shows Sys.LastLogs_Dat[0]
rectangle at (260,70)-(571,91): text "%s"; shows Sys.LastLogs_Dat[1]
rectangle at (260,90)-(571,111): text "%s"; shows Sys.LastLogs_Dat[2]
rectangle at (260,110)-(571,131): text "%s"; shows Sys.LastLogs_Dat[3]
rectangle at (260,130)-(571,151): text "%s"; shows Sys.LastLogs_Dat[4]
rectangle at (260,150)-(571,171): text "%s"; shows Sys.LastLogs_Dat[5]
rectangle at (100,70)-(181,101): text "ALARM"; alarm colour if Sys.Alarm; runs INTERN ASSIGN Mode_Manual:=(FALSE)
rectangle at (100,30)-(181,61): text "WARNING"; alarm colour if Sys.Warning; runs INTERN ASSIGN Mode_Manual:=(TRUE)
button at (30,110)-(181,131): text "REARM"; runs INTERN ASSIGN Sys.Alarm:=(FALSE);INTERN ASSIGN Sys.Warning:=(FALSE)
button at (60,250)-(141,271): text "ANZ01"
rectangle at (260,30)-(771,51): text "Last error logs"
button at (60,280)-(141,301): text "ANZ02"
rectangle at (150,220)-(191,241): text "V"
rectangle at (230,220)-(281,241): text "P(kW)"
rectangle at (280,220)-(331,241): text "PF"
rectangle at (330,220)-(401,241): text "E(kWh)"
rectangle at (190,220)-(231,241): text "I(A)"
rectangle at (150,250)-(191,271): text "%d"; shows ANZ01.Data.V_3P/1000
rectangle at (190,250)-(231,271): text "%1.1f"; shows DWORD_TO_REAL(ANZ01.Data.I_3P)/1000
rectangle at (230,250)-(281,271): text "%1.1f"; shows DWORD_TO_REAL(ANZ01.Data.P_3P)/1000
rectangle at (280,250)-(331,271): text "%1.3f"; shows DINT_TO_REAL(ANZ01.Data.PF_3P)/1000
rectangle at (330,250)-(401,271): text "%d"; shows ANZ01.WH_3P/10
rectangle at (150,280)-(191,301): text "%d"; shows ANZ02.Data.V_3P/1000
rectangle at (190,280)-(231,301): text "%1.1f"; shows DWORD_TO_REAL(ANZ02.Data.I_3P)/1000
rectangle at (230,280)-(281,301): text "%1.1f"; shows DWORD_TO_REAL(ANZ02.Data.P_3P)/1000
rectangle at (280,280)-(331,301): text "%1.3f"; shows DINT_TO_REAL(ANZ02.Data.PF_3P)/1000
rectangle at (330,280)-(401,301): text "%d"; shows ANZ02.WH_3P/10
button at (430,250)-(511,271): text "HVAC01"
button at (430,280)-(511,301): text "HVAC02"
button at (490,450)-(561,471): text "LEARN 01"; runs INTERN ASSIGN DAI01.Status:=(1)
button at (670,450)-(741,471): text "LEARN 02"; runs INTERN ASSIGN DAI02.Status:=(1)
rectangle at (430,450)-(491,471): text "AID01"
rectangle at (610,450)-(671,471): text "AID02"
button at (60,350)-(141,371): text "ZTHL01"
button at (60,380)-(141,401): text "ZTHL02"
button at (60,410)-(141,431): text "ZTHL03"
button at (60,440)-(141,461): text "ZTHL04"
rectangle at (150,350)-(191,371): text "%1.1f"; shows INT_TO_REAL(ZTHL01.OUT_TEMP)/10
rectangle at (150,320)-(201,341): text "T [°C]"
rectangle at (200,320)-(251,341): text "RH [%]"
rectangle at (250,320)-(301,341): text "FLUX [lx]"
rectangle at (300,320)-(361,341): text "VBATT [V]"
rectangle at (360,320)-(401,341): text "LQI"
rectangle at (210,350)-(251,371): text "%d"; shows ZTHL01.OUT_HYGRO
rectangle at (260,350)-(301,371): text "%d"; shows ZTHL01.OUT_LUX
rectangle at (310,350)-(351,371): text "%1.2f"; shows INT_TO_REAL(ZTHL01.OUT_VBATT)/100
rectangle at (360,350)-(401,371): text "%d"; shows ZTHL01.OUT_LQI
rectangle at (150,380)-(191,401): text "%1.1f"; shows INT_TO_REAL(ZTHL02.OUT_TEMP)/10
rectangle at (210,380)-(251,401): text "%d"; shows ZTHL02.OUT_HYGRO
rectangle at (260,380)-(301,401): text "%d"; shows ZTHL02.OUT_LUX
rectangle at (310,380)-(351,401): text "%1.2f"; shows INT_TO_REAL(ZTHL02.OUT_VBATT)/100
rectangle at (360,380)-(401,401): text "%d"; shows ZTHL02.OUT_LQI
rectangle at (150,410)-(191,431): text "%1.1f"; shows INT_TO_REAL(ZTHL03.OUT_TEMP)/10
rectangle at (210,410)-(251,431): text "%d"; shows ZTHL03.OUT_HYGRO
rectangle at (260,410)-(301,431): text "%d"; shows ZTHL03.OUT_LUX
rectangle at (310,410)-(351,431): text "%1.2f"; shows INT_TO_REAL(ZTHL03.OUT_VBATT)/100
rectangle at (360,410)-(401,431): text "%d"; shows ZTHL03.OUT_LQI
rectangle at (150,440)-(191,461): text "%1.1f"; shows INT_TO_REAL(ZTHL04.OUT_TEMP)/10
rectangle at (210,440)-(251,461): text "%d"; shows ZTHL04.OUT_HYGRO
rectangle at (260,440)-(301,461): text "%d"; shows ZTHL04.OUT_LUX
rectangle at (310,440)-(351,461): text "%1.2f"; shows INT_TO_REAL(ZTHL04.OUT_VBATT)/100
rectangle at (360,440)-(401,461): text "%d"; shows ZTHL04.OUT_LQI
polygon at (410,320)-(760,340): text "LUX FEEDBACK"
rectangle at (430,350)-(441,371): alarm colour if DAI01.OutOfRange
rectangle at (430,380)-(441,401): alarm colour if DAI01.OutOfRange
rectangle at (430,410)-(441,431): alarm colour if DAI01.OutOfRange
rectangle at (610,350)-(621,371): alarm colour if DAI02.OutOfRange
rectangle at (610,380)-(621,401): alarm colour if DAI02.OutOfRange
rectangle at (610,410)-(621,431): alarm colour if DAI02.OutOfRange
button at (50,510)-(111,541): text "Chrono"; opens VIS_CHRONOEDITOR
rectangle at (520,220)-(601,241): text "SP Cold [°C]"
rectangle at (520,250)-(601,271): text "%1.1f"; shows WORD_TO_REAL(HVAC01.Data.ReadSetPointCold)/10
rectangle at (600,250)-(681,271): text "%1.1f"; shows WORD_TO_REAL(HVAC01.Data.ReadSetPointTemp)/10
rectangle at (680,250)-(761,271): text "%1.1f"; shows WORD_TO_REAL(HVAC01.Data.ReadSetPointHeat)/10
rectangle at (520,280)-(601,301): text "%1.1f"; shows WORD_TO_REAL(HVAC02.Data.ReadSetPointCold)/10
rectangle at (600,280)-(681,301): text "%1.1f"; shows WORD_TO_REAL(HVAC02.Data.ReadSetPointTemp)/10
rectangle at (680,280)-(761,301): text "%1.1f"; shows WORD_TO_REAL(HVAC02.Data.ReadSetPointHeat)/10
rectangle at (600,220)-(681,241): text "SP Temp [°C]"
rectangle at (680,220)-(761,241): text "SP Heat [°C]"
rectangle at (560,510)-(771,531): text "%s"; shows Sys.Time_LogString
16 more shapes without text or variables
17 elements of other kinds (tables, trends, ...) not read
*)

(* Visualisation VIS_CHRONOEDITOR
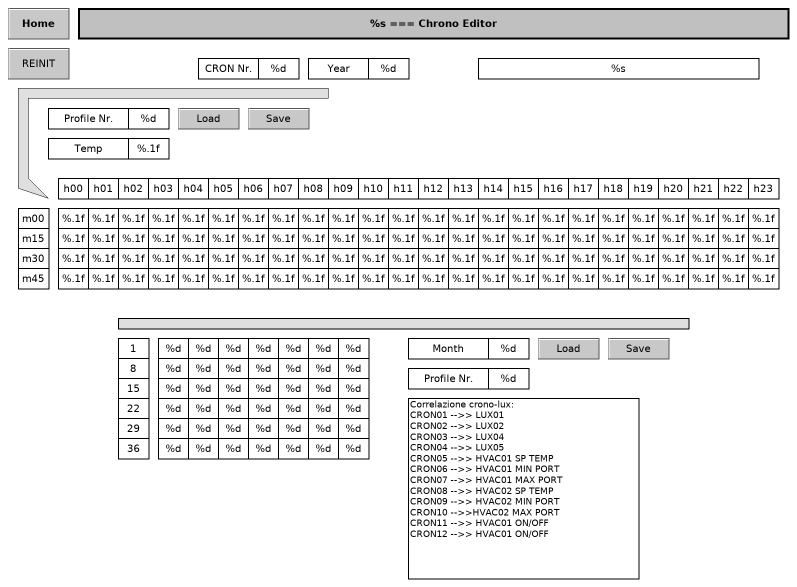
rectangle at (200,60)-(261,81): text "CRON Nr."
rectangle at (260,60)-(301,81): text "%d"; shows CronEd.CN_Sel; alarm colour if CronEd.CN_Sel<>CronEd.CN_Act; editable 1..12
rectangle at (50,110)-(131,131): text "Profile Nr."
rectangle at (130,110)-(171,131): text "%d"; shows CronEd.PR_Sel; alarm colour if CronEd.PR_Sel<>CronEd.PR_Act; editable 1..10
rectangle at (50,140)-(131,161): text "Temp"
rectangle at (130,140)-(171,161): text "%.1f"; shows CronEd.PR_TT; editable
button at (180,110)-(241,131): text "Load"; toggles CronEd.PR_Load
button at (250,110)-(311,131): text "Save"; toggles CronEd.PR_Save
rectangle at (20,210)-(51,231): text "m00"
rectangle at (20,230)-(51,251): text "m15"
rectangle at (20,250)-(51,271): text "m30"
rectangle at (20,270)-(51,291): text "m45"
rectangle at (80,10)-(791,41): text "%s === Chrono Editor"; shows .Plant_NAME
button at (10,10)-(71,41): text "Home"; opens PLC_VISU
rounded rectangle at (60,210)-(91,231): text "%.1f"; shows WORD_TO_REAL(CronEd.PR.Setpoint[0])/10; runs INTERN ASSIGN CronEd.PR.Setpoint[0]:=(REAL_TO_WORD(CronEd.PR_TT*10))
rounded rectangle at (60,230)-(91,251): text "%.1f"; shows WORD_TO_REAL(CronEd.PR.Setpoint[1])/10; runs INTERN ASSIGN CronEd.PR.Setpoint[1]:=(REAL_TO_WORD(CronEd.PR_TT*10))
rounded rectangle at (60,250)-(91,271): text "%.1f"; shows WORD_TO_REAL(CronEd.PR.Setpoint[2])/10; runs INTERN ASSIGN CronEd.PR.Setpoint[2]:=(REAL_TO_WORD(CronEd.PR_TT*10))
rounded rectangle at (60,270)-(91,291): text "%.1f"; shows WORD_TO_REAL(CronEd.PR.Setpoint[3])/10; runs INTERN ASSIGN CronEd.PR.Setpoint[3]:=(REAL_TO_WORD(CronEd.PR_TT*10))
rectangle at (60,180)-(91,201): text "h00"; runs INTERN ASSIGN CronEd.PR.Setpoint[0]:=(REAL_TO_WORD(CronEd.PR_TT*10));INTERN ASSIGN CronEd.PR.Setpoint[1]:=(REAL_TO_WORD(CronEd.PR_TT*10));INTERN ASSIGN CronEd.PR.Setpoint[2]:=(REAL_TO_WORD(CronEd.PR_TT*10));INTERN ASSIGN CronEd.PR.Setpoint[3]:=(REAL_TO_WORD(CronEd.PR_TT*10))
rounded rectangle at (90,210)-(121,231): text "%.1f"; shows WORD_TO_REAL(CronEd.PR.Setpoint[4])/10; runs INTERN ASSIGN CronEd.PR.Setpoint[4]:=(REAL_TO_WORD(CronEd.PR_TT*10))
rounded rectangle at (90,230)-(121,251): text "%.1f"; shows WORD_TO_REAL(CronEd.PR.Setpoint[5])/10; runs INTERN ASSIGN CronEd.PR.Setpoint[5]:=(REAL_TO_WORD(CronEd.PR_TT*10))
rounded rectangle at (90,250)-(121,271): text "%.1f"; shows WORD_TO_REAL(CronEd.PR.Setpoint[6])/10; runs INTERN ASSIGN CronEd.PR.Setpoint[6]:=(REAL_TO_WORD(CronEd.PR_TT*10))
rounded rectangle at (90,270)-(121,291): text "%.1f"; shows WORD_TO_REAL(CronEd.PR.Setpoint[7])/10; runs INTERN ASSIGN CronEd.PR.Setpoint[7]:=(REAL_TO_WORD(CronEd.PR_TT*10))
rectangle at (90,180)-(121,201): text "h01"; runs INTERN ASSIGN CronEd.PR.Setpoint[4]:=(REAL_TO_WORD(CronEd.PR_TT*10));INTERN ASSIGN CronEd.PR.Setpoint[5]:=(REAL_TO_WORD(CronEd.PR_TT*10));INTERN ASSIGN CronEd.PR.Setpoint[6]:=(REAL_TO_WORD(CronEd.PR_TT*10));INTERN ASSIGN CronEd.PR.Setpoint[7]:=(REAL_TO_WORD(CronEd.PR_TT*10))
rounded rectangle at (120,210)-(151,231): text "%.1f"; shows WORD_TO_REAL(CronEd.PR.Setpoint[8])/10; runs INTERN ASSIGN CronEd.PR.Setpoint[8]:=(REAL_TO_WORD(CronEd.PR_TT*10))
rounded rectangle at (120,230)-(151,251): text "%.1f"; shows WORD_TO_REAL(CronEd.PR.Setpoint[9])/10; runs INTERN ASSIGN CronEd.PR.Setpoint[9]:=(REAL_TO_WORD(CronEd.PR_TT*10))
rounded rectangle at (120,250)-(151,271): text "%.1f"; shows WORD_TO_REAL(CronEd.PR.Setpoint[10])/10; runs INTERN ASSIGN CronEd.PR.Setpoint[10]:=(REAL_TO_WORD(CronEd.PR_TT*10))
rounded rectangle at (120,270)-(151,291): text "%.1f"; shows WORD_TO_REAL(CronEd.PR.Setpoint[11])/10; runs INTERN ASSIGN CronEd.PR.Setpoint[11]:=(REAL_TO_WORD(CronEd.PR_TT*10))
rectangle at (120,180)-(151,201): text "h02"; runs INTERN ASSIGN CronEd.PR.Setpoint[8]:=(REAL_TO_WORD(CronEd.PR_TT*10));INTERN ASSIGN CronEd.PR.Setpoint[9]:=(REAL_TO_WORD(CronEd.PR_TT*10));INTERN ASSIGN CronEd.PR.Setpoint[10]:=(REAL_TO_WORD(CronEd.PR_TT*10));INTERN ASSIGN CronEd.PR.Setpoint[11]:=(REAL_TO_WORD(CronEd.PR_TT*10))
rounded rectangle at (150,210)-(181,231): text "%.1f"; shows WORD_TO_REAL(CronEd.PR.Setpoint[12])/10; runs INTERN ASSIGN CronEd.PR.Setpoint[12]:=(REAL_TO_WORD(CronEd.PR_TT*10))
rounded rectangle at (150,230)-(181,251): text "%.1f"; shows WORD_TO_REAL(CronEd.PR.Setpoint[13])/10; runs INTERN ASSIGN CronEd.PR.Setpoint[13]:=(REAL_TO_WORD(CronEd.PR_TT*10))
rounded rectangle at (150,250)-(181,271): text "%.1f"; shows WORD_TO_REAL(CronEd.PR.Setpoint[14])/10; runs INTERN ASSIGN CronEd.PR.Setpoint[14]:=(REAL_TO_WORD(CronEd.PR_TT*10))
rounded rectangle at (150,270)-(181,291): text "%.1f"; shows WORD_TO_REAL(CronEd.PR.Setpoint[15])/10; runs INTERN ASSIGN CronEd.PR.Setpoint[15]:=(REAL_TO_WORD(CronEd.PR_TT*10))
rectangle at (150,180)-(181,201): text "h03"; runs INTERN ASSIGN CronEd.PR.Setpoint[15]:=(REAL_TO_WORD(CronEd.PR_TT*10));INTERN ASSIGN CronEd.PR.Setpoint[14]:=(REAL_TO_WORD(CronEd.PR_TT*10));INTERN ASSIGN CronEd.PR.Setpoint[13]:=(REAL_TO_WORD(CronEd.PR_TT*10));INTERN ASSIGN CronEd.PR.Setpoint[12]:=(REAL_TO_WORD(CronEd.PR_TT*10))
rounded rectangle at (180,210)-(211,231): text "%.1f"; shows WORD_TO_REAL(CronEd.PR.Setpoint[16])/10; runs INTERN ASSIGN CronEd.PR.Setpoint[16]:=(REAL_TO_WORD(CronEd.PR_TT*10))
rounded rectangle at (180,230)-(211,251): text "%.1f"; shows WORD_TO_REAL(CronEd.PR.Setpoint[17])/10; runs INTERN ASSIGN CronEd.PR.Setpoint[17]:=(REAL_TO_WORD(CronEd.PR_TT*10))
rounded rectangle at (180,250)-(211,271): text "%.1f"; shows WORD_TO_REAL(CronEd.PR.Setpoint[18])/10; runs INTERN ASSIGN CronEd.PR.Setpoint[18]:=(REAL_TO_WORD(CronEd.PR_TT*10))
rounded rectangle at (180,270)-(211,291): text "%.1f"; shows WORD_TO_REAL(CronEd.PR.Setpoint[19])/10; runs INTERN ASSIGN CronEd.PR.Setpoint[19]:=(REAL_TO_WORD(CronEd.PR_TT*10))
rectangle at (180,180)-(211,201): text "h04"; runs INTERN ASSIGN CronEd.PR.Setpoint[19]:=(REAL_TO_WORD(CronEd.PR_TT*10));INTERN ASSIGN CronEd.PR.Setpoint[18]:=(REAL_TO_WORD(CronEd.PR_TT*10));INTERN ASSIGN CronEd.PR.Setpoint[17]:=(REAL_TO_WORD(CronEd.PR_TT*10));INTERN ASSIGN CronEd.PR.Setpoint[16]:=(REAL_TO_WORD(CronEd.PR_TT*10))
rounded rectangle at (210,210)-(241,231): text "%.1f"; shows WORD_TO_REAL(CronEd.PR.Setpoint[20])/10; runs INTERN ASSIGN CronEd.PR.Setpoint[20]:=(REAL_TO_WORD(CronEd.PR_TT*10))
rounded rectangle at (210,230)-(241,251): text "%.1f"; shows WORD_TO_REAL(CronEd.PR.Setpoint[21])/10; runs INTERN ASSIGN CronEd.PR.Setpoint[21]:=(REAL_TO_WORD(CronEd.PR_TT*10))
rounded rectangle at (210,250)-(241,271): text "%.1f"; shows WORD_TO_REAL(CronEd.PR.Setpoint[22])/10; runs INTERN ASSIGN CronEd.PR.Setpoint[22]:=(REAL_TO_WORD(CronEd.PR_TT*10))
rounded rectangle at (210,270)-(241,291): text "%.1f"; shows WORD_TO_REAL(CronEd.PR.Setpoint[23])/10; runs INTERN ASSIGN CronEd.PR.Setpoint[23]:=(REAL_TO_WORD(CronEd.PR_TT*10))
rectangle at (210,180)-(241,201): text "h05"; runs INTERN ASSIGN CronEd.PR.Setpoint[23]:=(REAL_TO_WORD(CronEd.PR_TT*10));INTERN ASSIGN CronEd.PR.Setpoint[22]:=(REAL_TO_WORD(CronEd.PR_TT*10));INTERN ASSIGN CronEd.PR.Setpoint[21]:=(REAL_TO_WORD(CronEd.PR_TT*10));INTERN ASSIGN CronEd.PR.Setpoint[20]:=(REAL_TO_WORD(CronEd.PR_TT*10))
rounded rectangle at (240,210)-(271,231): text "%.1f"; shows WORD_TO_REAL(CronEd.PR.Setpoint[24])/10; runs INTERN ASSIGN CronEd.PR.Setpoint[24]:=(REAL_TO_WORD(CronEd.PR_TT*10))
rounded rectangle at (240,230)-(271,251): text "%.1f"; shows WORD_TO_REAL(CronEd.PR.Setpoint[25])/10; runs INTERN ASSIGN CronEd.PR.Setpoint[25]:=(REAL_TO_WORD(CronEd.PR_TT*10))
rounded rectangle at (240,250)-(271,271): text "%.1f"; shows WORD_TO_REAL(CronEd.PR.Setpoint[26])/10; runs INTERN ASSIGN CronEd.PR.Setpoint[26]:=(REAL_TO_WORD(CronEd.PR_TT*10))
rounded rectangle at (240,270)-(271,291): text "%.1f"; shows WORD_TO_REAL(CronEd.PR.Setpoint[27])/10; runs INTERN ASSIGN CronEd.PR.Setpoint[27]:=(REAL_TO_WORD(CronEd.PR_TT*10))
rectangle at (240,180)-(271,201): text "h06"; runs INTERN ASSIGN CronEd.PR.Setpoint[27]:=(REAL_TO_WORD(CronEd.PR_TT*10));INTERN ASSIGN CronEd.PR.Setpoint[26]:=(REAL_TO_WORD(CronEd.PR_TT*10));INTERN ASSIGN CronEd.PR.Setpoint[25]:=(REAL_TO_WORD(CronEd.PR_TT*10));INTERN ASSIGN CronEd.PR.Setpoint[24]:=(REAL_TO_WORD(CronEd.PR_TT*10))
rounded rectangle at (270,210)-(301,231): text "%.1f"; shows WORD_TO_REAL(CronEd.PR.Setpoint[28])/10; runs INTERN ASSIGN CronEd.PR.Setpoint[28]:=(REAL_TO_WORD(CronEd.PR_TT*10))
rounded rectangle at (270,230)-(301,251): text "%.1f"; shows WORD_TO_REAL(CronEd.PR.Setpoint[29])/10; runs INTERN ASSIGN CronEd.PR.Setpoint[29]:=(REAL_TO_WORD(CronEd.PR_TT*10))
rounded rectangle at (270,250)-(301,271): text "%.1f"; shows WORD_TO_REAL(CronEd.PR.Setpoint[30])/10; runs INTERN ASSIGN CronEd.PR.Setpoint[30]:=(REAL_TO_WORD(CronEd.PR_TT*10))
rounded rectangle at (270,270)-(301,291): text "%.1f"; shows WORD_TO_REAL(CronEd.PR.Setpoint[31])/10; runs INTERN ASSIGN CronEd.PR.Setpoint[31]:=(REAL_TO_WORD(CronEd.PR_TT*10))
rectangle at (270,180)-(301,201): text "h07"; runs INTERN ASSIGN CronEd.PR.Setpoint[31]:=(REAL_TO_WORD(CronEd.PR_TT*10));INTERN ASSIGN CronEd.PR.Setpoint[30]:=(REAL_TO_WORD(CronEd.PR_TT*10));INTERN ASSIGN CronEd.PR.Setpoint[29]:=(REAL_TO_WORD(CronEd.PR_TT*10));INTERN ASSIGN CronEd.PR.Setpoint[28]:=(REAL_TO_WORD(CronEd.PR_TT*10))
rounded rectangle at (300,210)-(331,231): text "%.1f"; shows WORD_TO_REAL(CronEd.PR.Setpoint[32])/10; runs INTERN ASSIGN CronEd.PR.Setpoint[32]:=(REAL_TO_WORD(CronEd.PR_TT*10))
rounded rectangle at (300,230)-(331,251): text "%.1f"; shows WORD_TO_REAL(CronEd.PR.Setpoint[33])/10; runs INTERN ASSIGN CronEd.PR.Setpoint[33]:=(REAL_TO_WORD(CronEd.PR_TT*10))
rounded rectangle at (300,250)-(331,271): text "%.1f"; shows WORD_TO_REAL(CronEd.PR.Setpoint[34])/10; runs INTERN ASSIGN CronEd.PR.Setpoint[34]:=(REAL_TO_WORD(CronEd.PR_TT*10))
rounded rectangle at (300,270)-(331,291): text "%.1f"; shows WORD_TO_REAL(CronEd.PR.Setpoint[35])/10; runs INTERN ASSIGN CronEd.PR.Setpoint[35]:=(REAL_TO_WORD(CronEd.PR_TT*10))
rectangle at (300,180)-(331,201): text "h08"; runs INTERN ASSIGN CronEd.PR.Setpoint[35]:=(REAL_TO_WORD(CronEd.PR_TT*10));INTERN ASSIGN CronEd.PR.Setpoint[34]:=(REAL_TO_WORD(CronEd.PR_TT*10));INTERN ASSIGN CronEd.PR.Setpoint[33]:=(REAL_TO_WORD(CronEd.PR_TT*10));INTERN ASSIGN CronEd.PR.Setpoint[32]:=(REAL_TO_WORD(CronEd.PR_TT*10))
rounded rectangle at (330,210)-(361,231): text "%.1f"; shows WORD_TO_REAL(CronEd.PR.Setpoint[36])/10; runs INTERN ASSIGN CronEd.PR.Setpoint[36]:=(REAL_TO_WORD(CronEd.PR_TT*10))
rounded rectangle at (330,230)-(361,251): text "%.1f"; shows WORD_TO_REAL(CronEd.PR.Setpoint[37])/10; runs INTERN ASSIGN CronEd.PR.Setpoint[37]:=(REAL_TO_WORD(CronEd.PR_TT*10))
rounded rectangle at (330,250)-(361,271): text "%.1f"; shows WORD_TO_REAL(CronEd.PR.Setpoint[38])/10; runs INTERN ASSIGN CronEd.PR.Setpoint[38]:=(REAL_TO_WORD(CronEd.PR_TT*10))
rounded rectangle at (330,270)-(361,291): text "%.1f"; shows WORD_TO_REAL(CronEd.PR.Setpoint[39])/10; runs INTERN ASSIGN CronEd.PR.Setpoint[39]:=(REAL_TO_WORD(CronEd.PR_TT*10))
rectangle at (330,180)-(361,201): text "h09"; runs INTERN ASSIGN CronEd.PR.Setpoint[39]:=(REAL_TO_WORD(CronEd.PR_TT*10));INTERN ASSIGN CronEd.PR.Setpoint[38]:=(REAL_TO_WORD(CronEd.PR_TT*10));INTERN ASSIGN CronEd.PR.Setpoint[37]:=(REAL_TO_WORD(CronEd.PR_TT*10));INTERN ASSIGN CronEd.PR.Setpoint[36]:=(REAL_TO_WORD(CronEd.PR_TT*10))
rounded rectangle at (360,210)-(391,231): text "%.1f"; shows WORD_TO_REAL(CronEd.PR.Setpoint[40])/10; runs INTERN ASSIGN CronEd.PR.Setpoint[40]:=(REAL_TO_WORD(CronEd.PR_TT*10))
rounded rectangle at (360,230)-(391,251): text "%.1f"; shows WORD_TO_REAL(CronEd.PR.Setpoint[41])/10; runs INTERN ASSIGN CronEd.PR.Setpoint[41]:=(REAL_TO_WORD(CronEd.PR_TT*10))
rounded rectangle at (360,250)-(391,271): text "%.1f"; shows WORD_TO_REAL(CronEd.PR.Setpoint[42])/10; runs INTERN ASSIGN CronEd.PR.Setpoint[42]:=(REAL_TO_WORD(CronEd.PR_TT*10))
rounded rectangle at (360,270)-(391,291): text "%.1f"; shows WORD_TO_REAL(CronEd.PR.Setpoint[43])/10; runs INTERN ASSIGN CronEd.PR.Setpoint[43]:=(REAL_TO_WORD(CronEd.PR_TT*10))
rectangle at (360,180)-(391,201): text "h10"; runs INTERN ASSIGN CronEd.PR.Setpoint[43]:=(REAL_TO_WORD(CronEd.PR_TT*10));INTERN ASSIGN CronEd.PR.Setpoint[42]:=(REAL_TO_WORD(CronEd.PR_TT*10));INTERN ASSIGN CronEd.PR.Setpoint[41]:=(REAL_TO_WORD(CronEd.PR_TT*10));INTERN ASSIGN CronEd.PR.Setpoint[40]:=(REAL_TO_WORD(CronEd.PR_TT*10))
rounded rectangle at (390,210)-(421,231): text "%.1f"; shows WORD_TO_REAL(CronEd.PR.Setpoint[44])/10; runs INTERN ASSIGN CronEd.PR.Setpoint[44]:=(REAL_TO_WORD(CronEd.PR_TT*10))
rounded rectangle at (390,230)-(421,251): text "%.1f"; shows WORD_TO_REAL(CronEd.PR.Setpoint[45])/10; runs INTERN ASSIGN CronEd.PR.Setpoint[45]:=(REAL_TO_WORD(CronEd.PR_TT*10))
rounded rectangle at (390,250)-(421,271): text "%.1f"; shows WORD_TO_REAL(CronEd.PR.Setpoint[46])/10; runs INTERN ASSIGN CronEd.PR.Setpoint[46]:=(REAL_TO_WORD(CronEd.PR_TT*10))
rounded rectangle at (390,270)-(421,291): text "%.1f"; shows WORD_TO_REAL(CronEd.PR.Setpoint[47])/10; runs INTERN ASSIGN CronEd.PR.Setpoint[47]:=(REAL_TO_WORD(CronEd.PR_TT*10))
rectangle at (390,180)-(421,201): text "h11"; runs INTERN ASSIGN CronEd.PR.Setpoint[47]:=(REAL_TO_WORD(CronEd.PR_TT*10));INTERN ASSIGN CronEd.PR.Setpoint[46]:=(REAL_TO_WORD(CronEd.PR_TT*10));INTERN ASSIGN CronEd.PR.Setpoint[45]:=(REAL_TO_WORD(CronEd.PR_TT*10));INTERN ASSIGN CronEd.PR.Setpoint[44]:=(REAL_TO_WORD(CronEd.PR_TT*10))
rounded rectangle at (420,210)-(451,231): text "%.1f"; shows WORD_TO_REAL(CronEd.PR.Setpoint[48])/10; runs INTERN ASSIGN CronEd.PR.Setpoint[48]:=(REAL_TO_WORD(CronEd.PR_TT*10))
rounded rectangle at (420,230)-(451,251): text "%.1f"; shows WORD_TO_REAL(CronEd.PR.Setpoint[49])/10; runs INTERN ASSIGN CronEd.PR.Setpoint[49]:=(REAL_TO_WORD(CronEd.PR_TT*10))
rounded rectangle at (420,250)-(451,271): text "%.1f"; shows WORD_TO_REAL(CronEd.PR.Setpoint[50])/10; runs INTERN ASSIGN CronEd.PR.Setpoint[50]:=(REAL_TO_WORD(CronEd.PR_TT*10))
rounded rectangle at (420,270)-(451,291): text "%.1f"; shows WORD_TO_REAL(CronEd.PR.Setpoint[51])/10; runs INTERN ASSIGN CronEd.PR.Setpoint[51]:=(REAL_TO_WORD(CronEd.PR_TT*10))
rectangle at (420,180)-(451,201): text "h12"; runs INTERN ASSIGN CronEd.PR.Setpoint[51]:=(REAL_TO_WORD(CronEd.PR_TT*10));INTERN ASSIGN CronEd.PR.Setpoint[50]:=(REAL_TO_WORD(CronEd.PR_TT*10));INTERN ASSIGN CronEd.PR.Setpoint[49]:=(REAL_TO_WORD(CronEd.PR_TT*10));INTERN ASSIGN CronEd.PR.Setpoint[48]:=(REAL_TO_WORD(CronEd.PR_TT*10))
rounded rectangle at (450,210)-(481,231): text "%.1f"; shows WORD_TO_REAL(CronEd.PR.Setpoint[52])/10; runs INTERN ASSIGN CronEd.PR.Setpoint[52]:=(REAL_TO_WORD(CronEd.PR_TT*10))
rounded rectangle at (450,230)-(481,251): text "%.1f"; shows WORD_TO_REAL(CronEd.PR.Setpoint[53])/10; runs INTERN ASSIGN CronEd.PR.Setpoint[53]:=(REAL_TO_WORD(CronEd.PR_TT*10))
rounded rectangle at (450,250)-(481,271): text "%.1f"; shows WORD_TO_REAL(CronEd.PR.Setpoint[54])/10; runs INTERN ASSIGN CronEd.PR.Setpoint[54]:=(REAL_TO_WORD(CronEd.PR_TT*10))
rounded rectangle at (450,270)-(481,291): text "%.1f"; shows WORD_TO_REAL(CronEd.PR.Setpoint[55])/10; runs INTERN ASSIGN CronEd.PR.Setpoint[55]:=(REAL_TO_WORD(CronEd.PR_TT*10))
rectangle at (450,180)-(481,201): text "h13"; runs INTERN ASSIGN CronEd.PR.Setpoint[55]:=(REAL_TO_WORD(CronEd.PR_TT*10));INTERN ASSIGN CronEd.PR.Setpoint[54]:=(REAL_TO_WORD(CronEd.PR_TT*10));INTERN ASSIGN CronEd.PR.Setpoint[53]:=(REAL_TO_WORD(CronEd.PR_TT*10));INTERN ASSIGN CronEd.PR.Setpoint[52]:=(REAL_TO_WORD(CronEd.PR_TT*10))
rounded rectangle at (480,210)-(511,231): text "%.1f"; shows WORD_TO_REAL(CronEd.PR.Setpoint[56])/10; runs INTERN ASSIGN CronEd.PR.Setpoint[56]:=(REAL_TO_WORD(CronEd.PR_TT*10))
rounded rectangle at (480,230)-(511,251): text "%.1f"; shows WORD_TO_REAL(CronEd.PR.Setpoint[57])/10; runs INTERN ASSIGN CronEd.PR.Setpoint[57]:=(REAL_TO_WORD(CronEd.PR_TT*10))
rounded rectangle at (480,250)-(511,271): text "%.1f"; shows WORD_TO_REAL(CronEd.PR.Setpoint[58])/10; runs INTERN ASSIGN CronEd.PR.Setpoint[58]:=(REAL_TO_WORD(CronEd.PR_TT*10))
rounded rectangle at (480,270)-(511,291): text "%.1f"; shows WORD_TO_REAL(CronEd.PR.Setpoint[59])/10; runs INTERN ASSIGN CronEd.PR.Setpoint[59]:=(REAL_TO_WORD(CronEd.PR_TT*10))
rectangle at (480,180)-(511,201): text "h14"; runs INTERN ASSIGN CronEd.PR.Setpoint[59]:=(REAL_TO_WORD(CronEd.PR_TT*10));INTERN ASSIGN CronEd.PR.Setpoint[58]:=(REAL_TO_WORD(CronEd.PR_TT*10));INTERN ASSIGN CronEd.PR.Setpoint[57]:=(REAL_TO_WORD(CronEd.PR_TT*10));INTERN ASSIGN CronEd.PR.Setpoint[56]:=(REAL_TO_WORD(CronEd.PR_TT*10))
rounded rectangle at (510,210)-(541,231): text "%.1f"; shows WORD_TO_REAL(CronEd.PR.Setpoint[60])/10; runs INTERN ASSIGN CronEd.PR.Setpoint[60]:=(REAL_TO_WORD(CronEd.PR_TT*10))
rounded rectangle at (510,230)-(541,251): text "%.1f"; shows WORD_TO_REAL(CronEd.PR.Setpoint[61])/10; runs INTERN ASSIGN CronEd.PR.Setpoint[61]:=(REAL_TO_WORD(CronEd.PR_TT*10))
rounded rectangle at (510,250)-(541,271): text "%.1f"; shows WORD_TO_REAL(CronEd.PR.Setpoint[62])/10; runs INTERN ASSIGN CronEd.PR.Setpoint[62]:=(REAL_TO_WORD(CronEd.PR_TT*10))
rounded rectangle at (510,270)-(541,291): text "%.1f"; shows WORD_TO_REAL(CronEd.PR.Setpoint[63])/10; runs INTERN ASSIGN CronEd.PR.Setpoint[63]:=(REAL_TO_WORD(CronEd.PR_TT*10))
rectangle at (510,180)-(541,201): text "h15"; runs INTERN ASSIGN CronEd.PR.Setpoint[63]:=(REAL_TO_WORD(CronEd.PR_TT*10));INTERN ASSIGN CronEd.PR.Setpoint[62]:=(REAL_TO_WORD(CronEd.PR_TT*10));INTERN ASSIGN CronEd.PR.Setpoint[61]:=(REAL_TO_WORD(CronEd.PR_TT*10));INTERN ASSIGN CronEd.PR.Setpoint[60]:=(REAL_TO_WORD(CronEd.PR_TT*10))
rounded rectangle at (540,210)-(571,231): text "%.1f"; shows WORD_TO_REAL(CronEd.PR.Setpoint[64])/10; runs INTERN ASSIGN CronEd.PR.Setpoint[64]:=(REAL_TO_WORD(CronEd.PR_TT*10))
rounded rectangle at (540,230)-(571,251): text "%.1f"; shows WORD_TO_REAL(CronEd.PR.Setpoint[65])/10; runs INTERN ASSIGN CronEd.PR.Setpoint[65]:=(REAL_TO_WORD(CronEd.PR_TT*10))
rounded rectangle at (540,250)-(571,271): text "%.1f"; shows WORD_TO_REAL(CronEd.PR.Setpoint[66])/10; runs INTERN ASSIGN CronEd.PR.Setpoint[66]:=(REAL_TO_WORD(CronEd.PR_TT*10))
rounded rectangle at (540,270)-(571,291): text "%.1f"; shows WORD_TO_REAL(CronEd.PR.Setpoint[67])/10; runs INTERN ASSIGN CronEd.PR.Setpoint[67]:=(REAL_TO_WORD(CronEd.PR_TT*10))
rectangle at (540,180)-(571,201): text "h16"; runs INTERN ASSIGN CronEd.PR.Setpoint[67]:=(REAL_TO_WORD(CronEd.PR_TT*10));INTERN ASSIGN CronEd.PR.Setpoint[66]:=(REAL_TO_WORD(CronEd.PR_TT*10));INTERN ASSIGN CronEd.PR.Setpoint[65]:=(REAL_TO_WORD(CronEd.PR_TT*10));INTERN ASSIGN CronEd.PR.Setpoint[64]:=(REAL_TO_WORD(CronEd.PR_TT*10))
rounded rectangle at (570,210)-(601,231): text "%.1f"; shows WORD_TO_REAL(CronEd.PR.Setpoint[68])/10; runs INTERN ASSIGN CronEd.PR.Setpoint[68]:=(REAL_TO_WORD(CronEd.PR_TT*10))
rounded rectangle at (570,230)-(601,251): text "%.1f"; shows WORD_TO_REAL(CronEd.PR.Setpoint[69])/10; runs INTERN ASSIGN CronEd.PR.Setpoint[69]:=(REAL_TO_WORD(CronEd.PR_TT*10))
rounded rectangle at (570,250)-(601,271): text "%.1f"; shows WORD_TO_REAL(CronEd.PR.Setpoint[70])/10; runs INTERN ASSIGN CronEd.PR.Setpoint[70]:=(REAL_TO_WORD(CronEd.PR_TT*10))
rounded rectangle at (570,270)-(601,291): text "%.1f"; shows WORD_TO_REAL(CronEd.PR.Setpoint[71])/10; runs INTERN ASSIGN CronEd.PR.Setpoint[71]:=(REAL_TO_WORD(CronEd.PR_TT*10))
rectangle at (570,180)-(601,201): text "h17"; runs INTERN ASSIGN CronEd.PR.Setpoint[71]:=(REAL_TO_WORD(CronEd.PR_TT*10));INTERN ASSIGN CronEd.PR.Setpoint[70]:=(REAL_TO_WORD(CronEd.PR_TT*10));INTERN ASSIGN CronEd.PR.Setpoint[69]:=(REAL_TO_WORD(CronEd.PR_TT*10));INTERN ASSIGN CronEd.PR.Setpoint[68]:=(REAL_TO_WORD(CronEd.PR_TT*10))
rounded rectangle at (600,210)-(631,231): text "%.1f"; shows WORD_TO_REAL(CronEd.PR.Setpoint[72])/10; runs INTERN ASSIGN CronEd.PR.Setpoint[72]:=(REAL_TO_WORD(CronEd.PR_TT*10))
rounded rectangle at (600,230)-(631,251): text "%.1f"; shows WORD_TO_REAL(CronEd.PR.Setpoint[73])/10; runs INTERN ASSIGN CronEd.PR.Setpoint[73]:=(REAL_TO_WORD(CronEd.PR_TT*10))
rounded rectangle at (600,250)-(631,271): text "%.1f"; shows WORD_TO_REAL(CronEd.PR.Setpoint[74])/10; runs INTERN ASSIGN CronEd.PR.Setpoint[74]:=(REAL_TO_WORD(CronEd.PR_TT*10))
rounded rectangle at (600,270)-(631,291): text "%.1f"; shows WORD_TO_REAL(CronEd.PR.Setpoint[75])/10; runs INTERN ASSIGN CronEd.PR.Setpoint[75]:=(REAL_TO_WORD(CronEd.PR_TT*10))
rectangle at (600,180)-(631,201): text "h18"; runs INTERN ASSIGN CronEd.PR.Setpoint[75]:=(REAL_TO_WORD(CronEd.PR_TT*10));INTERN ASSIGN CronEd.PR.Setpoint[74]:=(REAL_TO_WORD(CronEd.PR_TT*10));INTERN ASSIGN CronEd.PR.Setpoint[73]:=(REAL_TO_WORD(CronEd.PR_TT*10));INTERN ASSIGN CronEd.PR.Setpoint[72]:=(REAL_TO_WORD(CronEd.PR_TT*10))
rounded rectangle at (630,210)-(661,231): text "%.1f"; shows WORD_TO_REAL(CronEd.PR.Setpoint[76])/10; runs INTERN ASSIGN CronEd.PR.Setpoint[76]:=(REAL_TO_WORD(CronEd.PR_TT*10))
rounded rectangle at (630,230)-(661,251): text "%.1f"; shows WORD_TO_REAL(CronEd.PR.Setpoint[77])/10; runs INTERN ASSIGN CronEd.PR.Setpoint[77]:=(REAL_TO_WORD(CronEd.PR_TT*10))
rounded rectangle at (630,250)-(661,271): text "%.1f"; shows WORD_TO_REAL(CronEd.PR.Setpoint[78])/10; runs INTERN ASSIGN CronEd.PR.Setpoint[78]:=(REAL_TO_WORD(CronEd.PR_TT*10))
rounded rectangle at (630,270)-(661,291): text "%.1f"; shows WORD_TO_REAL(CronEd.PR.Setpoint[79])/10; runs INTERN ASSIGN CronEd.PR.Setpoint[79]:=(REAL_TO_WORD(CronEd.PR_TT*10))
rectangle at (630,180)-(661,201): text "h19"; runs INTERN ASSIGN CronEd.PR.Setpoint[79]:=(REAL_TO_WORD(CronEd.PR_TT*10));INTERN ASSIGN CronEd.PR.Setpoint[78]:=(REAL_TO_WORD(CronEd.PR_TT*10));INTERN ASSIGN CronEd.PR.Setpoint[77]:=(REAL_TO_WORD(CronEd.PR_TT*10));INTERN ASSIGN CronEd.PR.Setpoint[76]:=(REAL_TO_WORD(CronEd.PR_TT*10))
rounded rectangle at (660,210)-(691,231): text "%.1f"; shows WORD_TO_REAL(CronEd.PR.Setpoint[80])/10; runs INTERN ASSIGN CronEd.PR.Setpoint[80]:=(REAL_TO_WORD(CronEd.PR_TT*10))
rounded rectangle at (660,230)-(691,251): text "%.1f"; shows WORD_TO_REAL(CronEd.PR.Setpoint[81])/10; runs INTERN ASSIGN CronEd.PR.Setpoint[81]:=(REAL_TO_WORD(CronEd.PR_TT*10))
rounded rectangle at (660,250)-(691,271): text "%.1f"; shows WORD_TO_REAL(CronEd.PR.Setpoint[82])/10; runs INTERN ASSIGN CronEd.PR.Setpoint[82]:=(REAL_TO_WORD(CronEd.PR_TT*10))
rounded rectangle at (660,270)-(691,291): text "%.1f"; shows WORD_TO_REAL(CronEd.PR.Setpoint[83])/10; runs INTERN ASSIGN CronEd.PR.Setpoint[83]:=(REAL_TO_WORD(CronEd.PR_TT*10))
rectangle at (660,180)-(691,201): text "h20"; runs INTERN ASSIGN CronEd.PR.Setpoint[83]:=(REAL_TO_WORD(CronEd.PR_TT*10));INTERN ASSIGN CronEd.PR.Setpoint[82]:=(REAL_TO_WORD(CronEd.PR_TT*10));INTERN ASSIGN CronEd.PR.Setpoint[81]:=(REAL_TO_WORD(CronEd.PR_TT*10));INTERN ASSIGN CronEd.PR.Setpoint[80]:=(REAL_TO_WORD(CronEd.PR_TT*10))
rounded rectangle at (690,210)-(721,231): text "%.1f"; shows WORD_TO_REAL(CronEd.PR.Setpoint[84])/10; runs INTERN ASSIGN CronEd.PR.Setpoint[84]:=(REAL_TO_WORD(CronEd.PR_TT*10))
rounded rectangle at (690,230)-(721,251): text "%.1f"; shows WORD_TO_REAL(CronEd.PR.Setpoint[85])/10; runs INTERN ASSIGN CronEd.PR.Setpoint[85]:=(REAL_TO_WORD(CronEd.PR_TT*10))
rounded rectangle at (690,250)-(721,271): text "%.1f"; shows WORD_TO_REAL(CronEd.PR.Setpoint[86])/10; runs INTERN ASSIGN CronEd.PR.Setpoint[86]:=(REAL_TO_WORD(CronEd.PR_TT*10))
rounded rectangle at (690,270)-(721,291): text "%.1f"; shows WORD_TO_REAL(CronEd.PR.Setpoint[87])/10; runs INTERN ASSIGN CronEd.PR.Setpoint[87]:=(REAL_TO_WORD(CronEd.PR_TT*10))
rectangle at (690,180)-(721,201): text "h21"; runs INTERN ASSIGN CronEd.PR.Setpoint[87]:=(REAL_TO_WORD(CronEd.PR_TT*10));INTERN ASSIGN CronEd.PR.Setpoint[86]:=(REAL_TO_WORD(CronEd.PR_TT*10));INTERN ASSIGN CronEd.PR.Setpoint[85]:=(REAL_TO_WORD(CronEd.PR_TT*10));INTERN ASSIGN CronEd.PR.Setpoint[84]:=(REAL_TO_WORD(CronEd.PR_TT*10))
rounded rectangle at (720,210)-(751,231): text "%.1f"; shows WORD_TO_REAL(CronEd.PR.Setpoint[88])/10; runs INTERN ASSIGN CronEd.PR.Setpoint[88]:=(REAL_TO_WORD(CronEd.PR_TT*10))
rounded rectangle at (720,230)-(751,251): text "%.1f"; shows WORD_TO_REAL(CronEd.PR.Setpoint[89])/10; runs INTERN ASSIGN CronEd.PR.Setpoint[89]:=(REAL_TO_WORD(CronEd.PR_TT*10))
rounded rectangle at (720,250)-(751,271): text "%.1f"; shows WORD_TO_REAL(CronEd.PR.Setpoint[90])/10; runs INTERN ASSIGN CronEd.PR.Setpoint[90]:=(REAL_TO_WORD(CronEd.PR_TT*10))
rounded rectangle at (720,270)-(751,291): text "%.1f"; shows WORD_TO_REAL(CronEd.PR.Setpoint[91])/10; runs INTERN ASSIGN CronEd.PR.Setpoint[91]:=(REAL_TO_WORD(CronEd.PR_TT*10))
rectangle at (720,180)-(751,201): text "h22"; runs INTERN ASSIGN CronEd.PR.Setpoint[91]:=(REAL_TO_WORD(CronEd.PR_TT*10));INTERN ASSIGN CronEd.PR.Setpoint[90]:=(REAL_TO_WORD(CronEd.PR_TT*10));INTERN ASSIGN CronEd.PR.Setpoint[89]:=(REAL_TO_WORD(CronEd.PR_TT*10));INTERN ASSIGN CronEd.PR.Setpoint[88]:=(REAL_TO_WORD(CronEd.PR_TT*10))
rounded rectangle at (750,210)-(781,231): text "%.1f"; shows WORD_TO_REAL(CronEd.PR.Setpoint[92])/10; runs INTERN ASSIGN CronEd.PR.Setpoint[92]:=(REAL_TO_WORD(CronEd.PR_TT*10))
rounded rectangle at (750,230)-(781,251): text "%.1f"; shows WORD_TO_REAL(CronEd.PR.Setpoint[93])/10; runs INTERN ASSIGN CronEd.PR.Setpoint[93]:=(REAL_TO_WORD(CronEd.PR_TT*10))
rounded rectangle at (750,250)-(781,271): text "%.1f"; shows WORD_TO_REAL(CronEd.PR.Setpoint[94])/10; runs INTERN ASSIGN CronEd.PR.Setpoint[94]:=(REAL_TO_WORD(CronEd.PR_TT*10))
rounded rectangle at (750,270)-(781,291): text "%.1f"; shows WORD_TO_REAL(CronEd.PR.Setpoint[95])/10; runs INTERN ASSIGN CronEd.PR.Setpoint[95]:=(REAL_TO_WORD(CronEd.PR_TT*10))
rectangle at (750,180)-(781,201): text "h23"; runs INTERN ASSIGN CronEd.PR.Setpoint[95]:=(REAL_TO_WORD(CronEd.PR_TT*10));INTERN ASSIGN CronEd.PR.Setpoint[94]:=(REAL_TO_WORD(CronEd.PR_TT*10));INTERN ASSIGN CronEd.PR.Setpoint[93]:=(REAL_TO_WORD(CronEd.PR_TT*10));INTERN ASSIGN CronEd.PR.Setpoint[92]:=(REAL_TO_WORD(CronEd.PR_TT*10))
rectangle at (410,340)-(491,361): text "Month"
rectangle at (490,340)-(531,361): text "%d"; shows CronEd.CA_Sel; alarm colour if CronEd.CA_Sel<>CronEd.CA_Act; editable 1..12
rectangle at (410,370)-(491,391): text "Profile Nr."
rectangle at (490,370)-(531,391): text "%d"; shows CronEd.CA_TPR; editable 0..10
button at (540,340)-(601,361): text "Load"; toggles CronEd.CA_Load
button at (610,340)-(671,361): text "Save"; toggles CronEd.CA_Save
rounded rectangle at (160,340)-(191,361): text "%d"; shows CronEd.CA.Profile[0]; invisible if CronEd.CA_DayF>0; alarm colour if CronEd.CA.Profile[0]=0; runs INTERN ASSIGN CronEd.CA.Profile[0]:=(CronEd.CA_TPR)
rectangle at (120,340)-(151,361): text "1"
rounded rectangle at (190,340)-(221,361): text "%d"; shows CronEd.CA.Profile[1]; invisible if CronEd.CA_DayF>1; alarm colour if CronEd.CA.Profile[1]=0; runs INTERN ASSIGN CronEd.CA.Profile[1]:=(CronEd.CA_TPR)
rounded rectangle at (220,340)-(251,361): text "%d"; shows CronEd.CA.Profile[2]; invisible if CronEd.CA_DayF>2; alarm colour if CronEd.CA.Profile[2]=0; runs INTERN ASSIGN CronEd.CA.Profile[2]:=(CronEd.CA_TPR)
rounded rectangle at (250,340)-(281,361): text "%d"; shows CronEd.CA.Profile[3]; invisible if CronEd.CA_DayF>3; alarm colour if CronEd.CA.Profile[3]=0; runs INTERN ASSIGN CronEd.CA.Profile[3]:=(CronEd.CA_TPR)
rounded rectangle at (280,340)-(311,361): text "%d"; shows CronEd.CA.Profile[4]; invisible if CronEd.CA_DayF>4; alarm colour if CronEd.CA.Profile[4]=0; runs INTERN ASSIGN CronEd.CA.Profile[4]:=(CronEd.CA_TPR)
rounded rectangle at (310,340)-(341,361): text "%d"; shows CronEd.CA.Profile[5]; invisible if CronEd.CA_DayF>5; alarm colour if CronEd.CA.Profile[5]=0; runs INTERN ASSIGN CronEd.CA.Profile[5]:=(CronEd.CA_TPR)
rounded rectangle at (340,340)-(371,361): text "%d"; shows CronEd.CA.Profile[6]; alarm colour if CronEd.CA.Profile[6]=0; runs INTERN ASSIGN CronEd.CA.Profile[6]:=(CronEd.CA_TPR)
rounded rectangle at (160,360)-(191,381): text "%d"; shows CronEd.CA.Profile[7]; alarm colour if CronEd.CA.Profile[7]=0; runs INTERN ASSIGN CronEd.CA.Profile[7]:=(CronEd.CA_TPR)
rectangle at (120,360)-(151,381): text "8"
rounded rectangle at (190,360)-(221,381): text "%d"; shows CronEd.CA.Profile[8]; alarm colour if CronEd.CA.Profile[8]=0; runs INTERN ASSIGN CronEd.CA.Profile[8]:=(CronEd.CA_TPR)
rounded rectangle at (220,360)-(251,381): text "%d"; shows CronEd.CA.Profile[9]; alarm colour if CronEd.CA.Profile[9]=0; runs INTERN ASSIGN CronEd.CA.Profile[9]:=(CronEd.CA_TPR)
rounded rectangle at (250,360)-(281,381): text "%d"; shows CronEd.CA.Profile[10]; alarm colour if CronEd.CA.Profile[10]=0; runs INTERN ASSIGN CronEd.CA.Profile[10]:=(CronEd.CA_TPR)
rounded rectangle at (280,360)-(311,381): text "%d"; shows CronEd.CA.Profile[11]; alarm colour if CronEd.CA.Profile[11]=0; runs INTERN ASSIGN CronEd.CA.Profile[11]:=(CronEd.CA_TPR)
rounded rectangle at (310,360)-(341,381): text "%d"; shows CronEd.CA.Profile[12]; alarm colour if CronEd.CA.Profile[12]=0; runs INTERN ASSIGN CronEd.CA.Profile[12]:=(CronEd.CA_TPR)
rounded rectangle at (340,360)-(371,381): text "%d"; shows CronEd.CA.Profile[13]; alarm colour if CronEd.CA.Profile[13]=0; runs INTERN ASSIGN CronEd.CA.Profile[13]:=(CronEd.CA_TPR)
rounded rectangle at (160,380)-(191,401): text "%d"; shows CronEd.CA.Profile[14]; alarm colour if CronEd.CA.Profile[14]=0; runs INTERN ASSIGN CronEd.CA.Profile[14]:=(CronEd.CA_TPR)
rectangle at (120,380)-(151,401): text "15"
rounded rectangle at (190,380)-(221,401): text "%d"; shows CronEd.CA.Profile[15]; alarm colour if CronEd.CA.Profile[15]=0; runs INTERN ASSIGN CronEd.CA.Profile[15]:=(CronEd.CA_TPR)
rounded rectangle at (220,380)-(251,401): text "%d"; shows CronEd.CA.Profile[16]; alarm colour if CronEd.CA.Profile[16]=0; runs INTERN ASSIGN CronEd.CA.Profile[16]:=(CronEd.CA_TPR)
rounded rectangle at (250,380)-(281,401): text "%d"; shows CronEd.CA.Profile[17]; alarm colour if CronEd.CA.Profile[17]=0; runs INTERN ASSIGN CronEd.CA.Profile[17]:=(CronEd.CA_TPR)
rounded rectangle at (280,380)-(311,401): text "%d"; shows CronEd.CA.Profile[18]; alarm colour if CronEd.CA.Profile[18]=0; runs INTERN ASSIGN CronEd.CA.Profile[18]:=(CronEd.CA_TPR)
rounded rectangle at (310,380)-(341,401): text "%d"; shows CronEd.CA.Profile[19]; alarm colour if CronEd.CA.Profile[19]=0; runs INTERN ASSIGN CronEd.CA.Profile[19]:=(CronEd.CA_TPR)
rounded rectangle at (340,380)-(371,401): text "%d"; shows CronEd.CA.Profile[20]; alarm colour if CronEd.CA.Profile[20]=0; runs INTERN ASSIGN CronEd.CA.Profile[20]:=(CronEd.CA_TPR)
rounded rectangle at (160,400)-(191,421): text "%d"; shows CronEd.CA.Profile[21]; alarm colour if CronEd.CA.Profile[21]=0; runs INTERN ASSIGN CronEd.CA.Profile[21]:=(CronEd.CA_TPR)
rectangle at (120,400)-(151,421): text "22"
rounded rectangle at (190,400)-(221,421): text "%d"; shows CronEd.CA.Profile[22]; alarm colour if CronEd.CA.Profile[22]=0; runs INTERN ASSIGN CronEd.CA.Profile[22]:=(CronEd.CA_TPR)
rounded rectangle at (220,400)-(251,421): text "%d"; shows CronEd.CA.Profile[23]; alarm colour if CronEd.CA.Profile[23]=0; runs INTERN ASSIGN CronEd.CA.Profile[23]:=(CronEd.CA_TPR)
rounded rectangle at (250,400)-(281,421): text "%d"; shows CronEd.CA.Profile[24]; alarm colour if CronEd.CA.Profile[24]=0; runs INTERN ASSIGN CronEd.CA.Profile[24]:=(CronEd.CA_TPR)
rounded rectangle at (280,400)-(311,421): text "%d"; shows CronEd.CA.Profile[25]; alarm colour if CronEd.CA.Profile[25]=0; runs INTERN ASSIGN CronEd.CA.Profile[25]:=(CronEd.CA_TPR)
rounded rectangle at (310,400)-(341,421): text "%d"; shows CronEd.CA.Profile[26]; alarm colour if CronEd.CA.Profile[26]=0; runs INTERN ASSIGN CronEd.CA.Profile[26]:=(CronEd.CA_TPR)
rounded rectangle at (340,400)-(371,421): text "%d"; shows CronEd.CA.Profile[27]; alarm colour if CronEd.CA.Profile[27]=0; runs INTERN ASSIGN CronEd.CA.Profile[27]:=(CronEd.CA_TPR)
rounded rectangle at (160,420)-(191,441): text "%d"; shows CronEd.CA.Profile[28]; alarm colour if CronEd.CA.Profile[28]=0; runs INTERN ASSIGN CronEd.CA.Profile[28]:=(CronEd.CA_TPR)
rectangle at (120,420)-(151,441): text "29"
rounded rectangle at (190,420)-(221,441): text "%d"; shows CronEd.CA.Profile[29]; alarm colour if CronEd.CA.Profile[29]=0; runs INTERN ASSIGN CronEd.CA.Profile[29]:=(CronEd.CA_TPR)
rounded rectangle at (220,420)-(251,441): text "%d"; shows CronEd.CA.Profile[30]; alarm colour if CronEd.CA.Profile[30]=0; runs INTERN ASSIGN CronEd.CA.Profile[30]:=(CronEd.CA_TPR)
rounded rectangle at (250,420)-(281,441): text "%d"; shows CronEd.CA.Profile[31]; alarm colour if CronEd.CA.Profile[31]=0; runs INTERN ASSIGN CronEd.CA.Profile[31]:=(CronEd.CA_TPR)
rounded rectangle at (280,420)-(311,441): text "%d"; shows CronEd.CA.Profile[32]; invisible if CronEd.CA_DayL<32; alarm colour if CronEd.CA.Profile[32]=0; runs INTERN ASSIGN CronEd.CA.Profile[32]:=(CronEd.CA_TPR)
rounded rectangle at (310,420)-(341,441): text "%d"; shows CronEd.CA.Profile[33]; invisible if CronEd.CA_DayL<33; alarm colour if CronEd.CA.Profile[33]=0; runs INTERN ASSIGN CronEd.CA.Profile[33]:=(CronEd.CA_TPR)
rounded rectangle at (340,420)-(371,441): text "%d"; shows CronEd.CA.Profile[34]; invisible if CronEd.CA_DayL<34; alarm colour if CronEd.CA.Profile[34]=0; runs INTERN ASSIGN CronEd.CA.Profile[34]:=(CronEd.CA_TPR)
rounded rectangle at (160,440)-(191,461): text "%d"; shows CronEd.CA.Profile[35]; invisible if CronEd.CA_DayL<35; alarm colour if CronEd.CA.Profile[35]=0; runs INTERN ASSIGN CronEd.CA.Profile[35]:=(CronEd.CA_TPR)
rectangle at (120,440)-(151,461): text "36"; invisible if CronEd.CA_DayL<35
rounded rectangle at (190,440)-(221,461): text "%d"; shows CronEd.CA.Profile[36]; invisible if CronEd.CA_DayL<36; alarm colour if CronEd.CA.Profile[36]=0; runs INTERN ASSIGN CronEd.CA.Profile[36]:=(CronEd.CA_TPR)
rounded rectangle at (220,440)-(251,461): text "%d"; shows CronEd.CA.Profile[37]; invisible if CronEd.CA_DayL<37; alarm colour if CronEd.CA.Profile[37]=0; runs INTERN ASSIGN CronEd.CA.Profile[37]:=(CronEd.CA_TPR)
rounded rectangle at (250,440)-(281,461): text "%d"; shows CronEd.CA.Profile[38]; invisible if CronEd.CA_DayL<38; alarm colour if CronEd.CA.Profile[38]=0; runs INTERN ASSIGN CronEd.CA.Profile[38]:=(CronEd.CA_TPR)
rounded rectangle at (280,440)-(311,461): text "%d"; shows CronEd.CA.Profile[39]; invisible if CronEd.CA_DayL<39; alarm colour if CronEd.CA.Profile[39]=0; runs INTERN ASSIGN CronEd.CA.Profile[39]:=(CronEd.CA_TPR)
rounded rectangle at (310,440)-(341,461): text "%d"; shows CronEd.CA.Profile[40]; invisible if CronEd.CA_DayL<40; alarm colour if CronEd.CA.Profile[40]=0; runs INTERN ASSIGN CronEd.CA.Profile[40]:=(CronEd.CA_TPR)
rounded rectangle at (340,440)-(371,461): text "%d"; shows CronEd.CA.Profile[41]; invisible if CronEd.CA_DayL<41; alarm colour if CronEd.CA.Profile[41]=0; runs INTERN ASSIGN CronEd.CA.Profile[41]:=(CronEd.CA_TPR)
rectangle at (310,60)-(371,81): text "Year"
rectangle at (370,60)-(411,81): text "%d"; shows CronEd.CN_YSel; alarm colour if CronEd.CN_YSel<>CronEd.CN_YAct; editable 2000..2100
rectangle at (480,60)-(761,81): text "%s"; shows CronEd.Message
button at (10,50)-(71,81): text "REINIT"; runs INTERN ASSIGN CRON01.InitOK:=(FALSE);INTERN ASSIGN CRON02.InitOK:=(FALSE);INTERN ASSIGN CRON03.InitOK:=(FALSE);INTERN ASSIGN CRON04.InitOK:=(FALSE);INTERN ASSIGN CRON05.InitOK:=(FALSE);INTERN ASSIGN CRON06.InitOK:=(FALSE)
rectangle at (410,400)-(641,581): text "Correlazione crono-lux: / CRON01 -->> LUX01 / CRON02 -->> LUX02 / CRON03 -->> LUX04 / CRON04 -->> LUX05 / CRON05 -->> HVAC01 SP TEMP / CRON06 -->> HVAC01 MIN PORT / CRON07 -->> HVAC01 MAX PORT / CRON08 -->> HVAC02 SP TEMP / CRON09 -->> HVAC02 MIN PORT / CRON10 -->>HVAC02 MAX PORT / CRON11 -->> HVAC01 ON/OFF / CRON12 -->> HVAC01 ON/OFF"
2 more shapes without text or variables
*)
